      A(    ;
      A     T    109;
      A     T    105;
      AN    I   1032.7;
      AN    M   1020.0;
      AN    M   1008.0;
      AN    M   1008.2;
      AN    M   1001.0;
      O     ;
      A(    ;
      O     I      0.7;
      O     I    180.4;
      )     ;
      AN    I   1032.0;
      )     ;
      A     M   1000.6;
      A     M   1500.6;
      AN    M   1020.3;
      AN    M   1030.0;
      AN    I   1032.5;
      =     Q   1032.6;
NETWORK
TITLE =

      A     I      0.1;
      =     Q   1032.7;
NETWORK
TITLE =

      A     I      0.0;
      A     M   1000.2;
      =     Q   1033.0;
NETWORK
TITLE =

      A     M   1000.6;
      A(    ;
      O     DB51.DBX  200.7;
      O     M   4000.6;
      )     ;
      A     I   1032.0;
      AN    I   1032.7;
      AN    M   1020.3;
      =     Q   1033.1;
NETWORK
TITLE =

      A     M   1000.6;
      A     M   1500.6;
      =     Q   1033.2;
NETWORK
TITLE =

      A     M   1001.7;
      A     M   1002.1;
      =     Q   1033.3;
NETWORK
TITLE =

      A     I   1041.5;
      =     Q   1033.5;
NETWORK
TITLE =

      A     I   1057.6;
      =     Q   1033.6;
NETWORK
TITLE =

      A     I   1049.7;
      =     Q   1033.7;
NETWORK
TITLE =

      A(    ;
      A     I    278.1;
      A     M   1054.0;
      A     M   1054.3;
      A     M   1051.0;
      A     M   1051.6;
      A     M   1052.0;
      A     M   1052.4;
      A     M   1052.6;
      A     M   1053.0;
      A     T    122;
      A     M    244.1;
      O     ;
      A     M   1042.0;
      A     M   1042.2;
      A     M   1042.4;
      A     M   1042.6;
      A     M   1043.2;
      A     M   1043.4;
      A     M   1044.4;
      A(    ;
      O     M   1040.6;
      O     M   1041.7;
      )     ;
      A     T    123;
      A     M    244.0;
      )     ;
      A     M   1009.4;
      A     M   1006.5;
      AN    M   1001.0;
      AN    M   1008.2;
      =     Q   1034.0;
NETWORK
TITLE =

      A     M   1512.5;
      A     M   1512.6;
      A     I    369.0;
      A     I    369.1;
      AN    Q    368.3;
      AN    Q   1034.5;
      =     Q   1034.4;
NETWORK
TITLE =

      A     M   1512.5;
      A     M   1512.6;
      AN    I    369.0;
      A     I    369.1;
      AN    Q    368.3;
      AN    Q   1034.4;
      =     Q   1034.5;
NETWORK
TITLE =
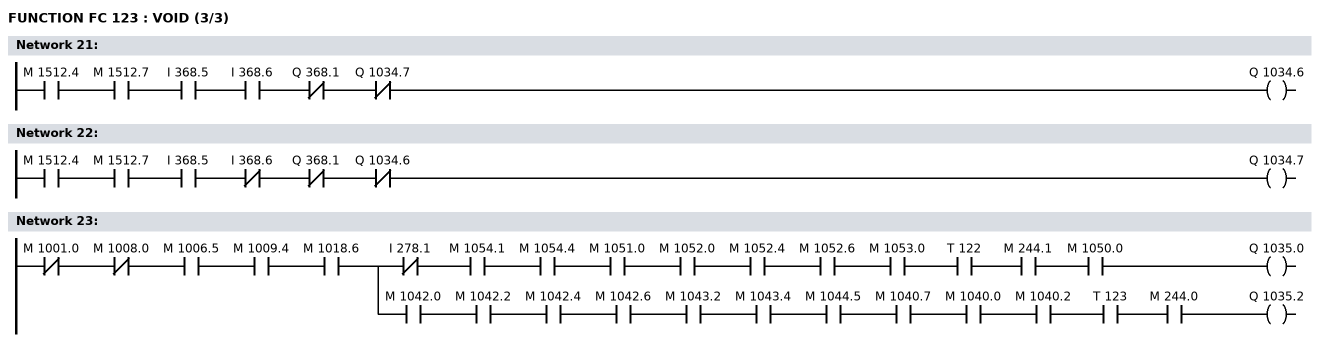

      A     M   1512.4;
      A     M   1512.7;
      A     I    368.5;
      A     I    368.6;
      AN    Q    368.1;
      AN    Q   1034.7;
      =     Q   1034.6;
NETWORK
TITLE =

      A     M   1512.4;
      A     M   1512.7;
      A     I    368.5;
      AN    I    368.6;
      AN    Q    368.1;
      AN    Q   1034.6;
      =     Q   1034.7;
NETWORK
TITLE =

      AN    M   1001.0;
      AN    M   1008.0;
      A     M   1006.5;
      A     M   1009.4;
      A     M   1018.6;
      =     L      0.0;
      A     L      0.0;
      AN    I    278.1;
      A     M   1054.1;
      A     M   1054.4;
      A     M   1051.0;
      A     M   1052.0;
      A     M   1052.4;
      A     M   1052.6;
      A     M   1053.0;
      A     T    122;
      A     M    244.1;
      A     M   1050.0;
      =     Q   1035.0;
      A     L      0.0;
      A     M   1042.0;
      A     M   1042.2;
      A     M   1042.4;
      A     M   1042.6;
      A     M   1043.2;
      A     M   1043.4;
      A     M   1044.5;
      A     M   1040.7;
      A     M   1040.0;
      A     M   1040.2;
      A     T    123;
      A     M    244.0;
      =     Q   1035.2;
END_FUNCTION

FUNCTION FC 124 : VOID
TITLE =
VERSION : 0.1

BEGIN
NETWORK
TITLE =
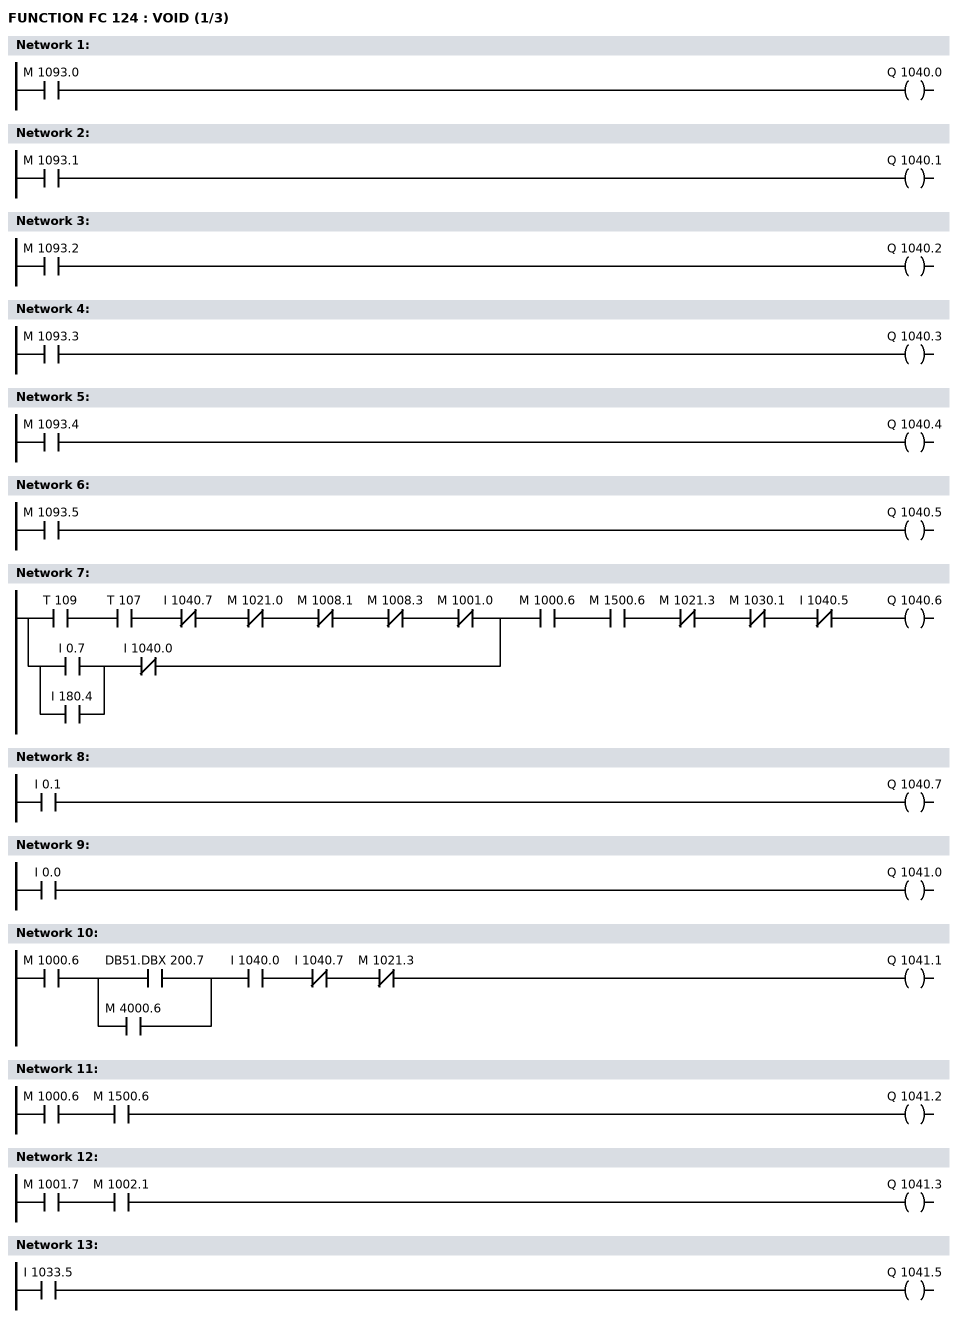

      A     M   1093.0;
      =     Q   1040.0;
NETWORK
TITLE =

      A     M   1093.1;
      =     Q   1040.1;
NETWORK
TITLE =

      A     M   1093.2;
      =     Q   1040.2;
NETWORK
TITLE =

      A     M   1093.3;
      =     Q   1040.3;
NETWORK
TITLE =

      A     M   1093.4;
      =     Q   1040.4;
NETWORK
TITLE =

      A     M   1093.5;
      =     Q   1040.5;
NETWORK
TITLE =

      A(    ;
      A     T    109;
      A     T    107;
      AN    I   1040.7;
      AN    M   1021.0;
      AN    M   1008.1;
      AN    M   1008.3;
      AN    M   1001.0;
      O     ;
      A(    ;
      O     I      0.7;
      O     I    180.4;
      )     ;
      AN    I   1040.0;
      )     ;
      A     M   1000.6;
      A     M   1500.6;
      AN    M   1021.3;
      AN    M   1030.1;
      AN    I   1040.5;
      =     Q   1040.6;
NETWORK
TITLE =

      A     I      0.1;
      =     Q   1040.7;
NETWORK
TITLE =

      A     I      0.0;
      =     Q   1041.0;
NETWORK
TITLE =

      A     M   1000.6;
      A(    ;
      O     DB51.DBX  200.7;
      O     M   4000.6;
      )     ;
      A     I   1040.0;
      AN    I   1040.7;
      AN    M   1021.3;
      =     Q   1041.1;
NETWORK
TITLE =

      A     M   1000.6;
      A     M   1500.6;
      =     Q   1041.2;
NETWORK
TITLE =

      A     M   1001.7;
      A     M   1002.1;
      =     Q   1041.3;
NETWORK
TITLE =

      A     I   1033.5;
      =     Q   1041.5;
NETWORK
TITLE =
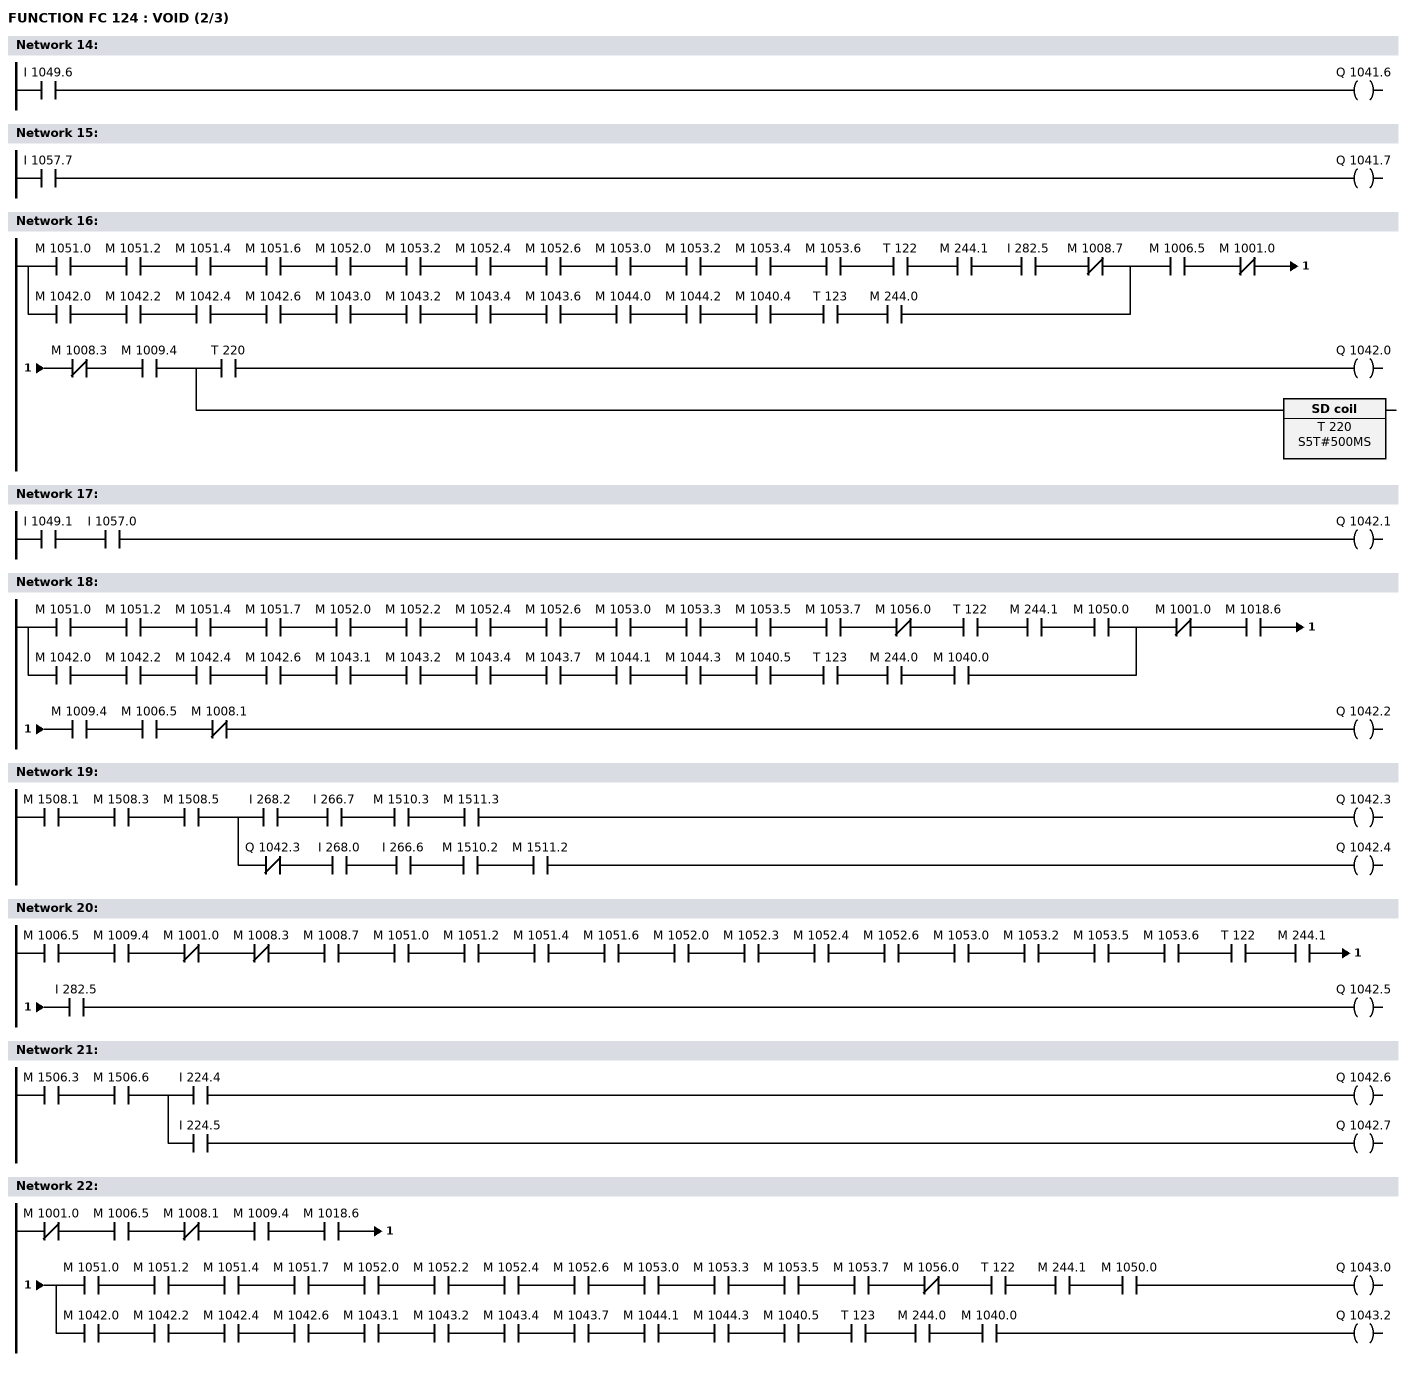

      A     I   1049.6;
      =     Q   1041.6;
NETWORK
TITLE =

      A     I   1057.7;
      =     Q   1041.7;
NETWORK
TITLE =

      A(    ;
      A     M   1051.0;
      A     M   1051.2;
      A     M   1051.4;
      A     M   1051.6;
      A     M   1052.0;
      A     M   1053.2;
      A     M   1052.4;
      A     M   1052.6;
      A     M   1053.0;
      A     M   1053.2;
      A     M   1053.4;
      A     M   1053.6;
      A     T    122;
      A     M    244.1;
      A     I    282.5;
      AN    M   1008.7;
      O     ;
      A     M   1042.0;
      A     M   1042.2;
      A     M   1042.4;
      A     M   1042.6;
      A     M   1043.0;
      A     M   1043.2;
      A     M   1043.4;
      A     M   1043.6;
      A     M   1044.0;
      A     M   1044.2;
      A     M   1040.4;
      A     T    123;
      A     M    244.0;
      )     ;
      A     M   1006.5;
      AN    M   1001.0;
      AN    M   1008.3;
      A     M   1009.4;
      =     L      0.0;
      A     L      0.0;
      A     T    220;
      =     Q   1042.0;
      A     L      0.0;
      BLD   102;
      L     S5T#500MS;
      SD    T    220;
NETWORK
TITLE =

      A     I   1049.1;
      A     I   1057.0;
      =     Q   1042.1;
NETWORK
TITLE =

      A(    ;
      A     M   1051.0;
      A     M   1051.2;
      A     M   1051.4;
      A     M   1051.7;
      A     M   1052.0;
      A     M   1052.2;
      A     M   1052.4;
      A     M   1052.6;
      A     M   1053.0;
      A     M   1053.3;
      A     M   1053.5;
      A     M   1053.7;
      AN    M   1056.0;
      A     T    122;
      A     M    244.1;
      A     M   1050.0;
      O     ;
      A     M   1042.0;
      A     M   1042.2;
      A     M   1042.4;
      A     M   1042.6;
      A     M   1043.1;
      A     M   1043.2;
      A     M   1043.4;
      A     M   1043.7;
      A     M   1044.1;
      A     M   1044.3;
      A     M   1040.5;
      A     T    123;
      A     M    244.0;
      A     M   1040.0;
      )     ;
      AN    M   1001.0;
      A     M   1018.6;
      A     M   1009.4;
      A     M   1006.5;
      AN    M   1008.1;
      =     Q   1042.2;
NETWORK
TITLE =

      A     M   1508.1;
      A     M   1508.3;
      A     M   1508.5;
      =     L      0.0;
      A     L      0.0;
      A     I    268.2;
      A     I    266.7;
      A     M   1510.3;
      A     M   1511.3;
      =     Q   1042.3;
      A     L      0.0;
      AN    Q   1042.3;
      A     I    268.0;
      A     I    266.6;
      A     M   1510.2;
      A     M   1511.2;
      =     Q   1042.4;
NETWORK
TITLE =

      A     M   1006.5;
      A     M   1009.4;
      AN    M   1001.0;
      AN    M   1008.3;
      A     M   1008.7;
      A     M   1051.0;
      A     M   1051.2;
      A     M   1051.4;
      A     M   1051.6;
      A     M   1052.0;
      A     M   1052.3;
      A     M   1052.4;
      A     M   1052.6;
      A     M   1053.0;
      A     M   1053.2;
      A     M   1053.5;
      A     M   1053.6;
      A     T    122;
      A     M    244.1;
      A     I    282.5;
      =     Q   1042.5;
NETWORK
TITLE =

      A     M   1506.3;
      A     M   1506.6;
      =     L      0.0;
      A     L      0.0;
      A     I    224.4;
      =     Q   1042.6;
      A     L      0.0;
      A     I    224.5;
      =     Q   1042.7;
NETWORK
TITLE =

      AN    M   1001.0;
      A     M   1006.5;
      AN    M   1008.1;
      A     M   1009.4;
      A     M   1018.6;
      =     L      0.0;
      A     L      0.0;
      A     M   1051.0;
      A     M   1051.2;
      A     M   1051.4;
      A     M   1051.7;
      A     M   1052.0;
      A     M   1052.2;
      A     M   1052.4;
      A     M   1052.6;
      A     M   1053.0;
      A     M   1053.3;
      A     M   1053.5;
      A     M   1053.7;
      AN    M   1056.0;
      A     T    122;
      A     M    244.1;
      A     M   1050.0;
      =     Q   1043.0;
      A     L      0.0;
      A     M   1042.0;
      A     M   1042.2;
      A     M   1042.4;
      A     M   1042.6;
      A     M   1043.1;
      A     M   1043.2;
      A     M   1043.4;
      A     M   1043.7;
      A     M   1044.1;
      A     M   1044.3;
      A     M   1040.5;
      A     T    123;
      A     M    244.0;
      A     M   1040.0;
      =     Q   1043.2;
NETWORK
TITLE =
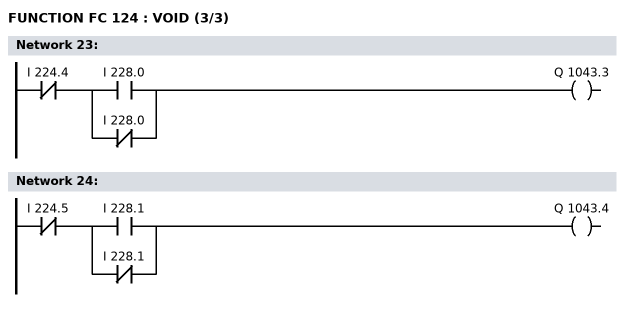

      AN    I    224.4;
      A(    ;
      O     I    228.0;
      ON    I    228.0;
      )     ;
      =     Q   1043.3;
NETWORK
TITLE =

      AN    I    224.5;
      A(    ;
      O     I    228.1;
      ON    I    228.1;
      )     ;
      =     Q   1043.4;
END_FUNCTION

FUNCTION FC 125 : VOID
TITLE =
VERSION : 0.1

BEGIN
NETWORK
TITLE =

      A     I   1048.0;
      JNB   _001;
      L     0;
      T     MB  1094;
_001: NOP   0;
NETWORK
TITLE =

      AN    OV;
      =     L      0.0;
      A     L      0.0;
      A     M    164.1;
      =     L      0.1;
      A     L      0.1;
      AN    M    167.7;
      A     I   1048.0;
      JNB   _002;
      L     11;
      T     MB  1094;
_002: NOP   0;
      A     L      0.1;
      A     M    167.7;
      A     I   1048.0;
      JNB   _003;
      L     19;
      T     MB  1094;
_003: NOP   0;
      A     L      0.0;
      A     M    164.0;
      A     I   1048.0;
      JNB   _004;
      L     1;
      T     MB  1094;
_004: NOP   0;
NETWORK
TITLE =
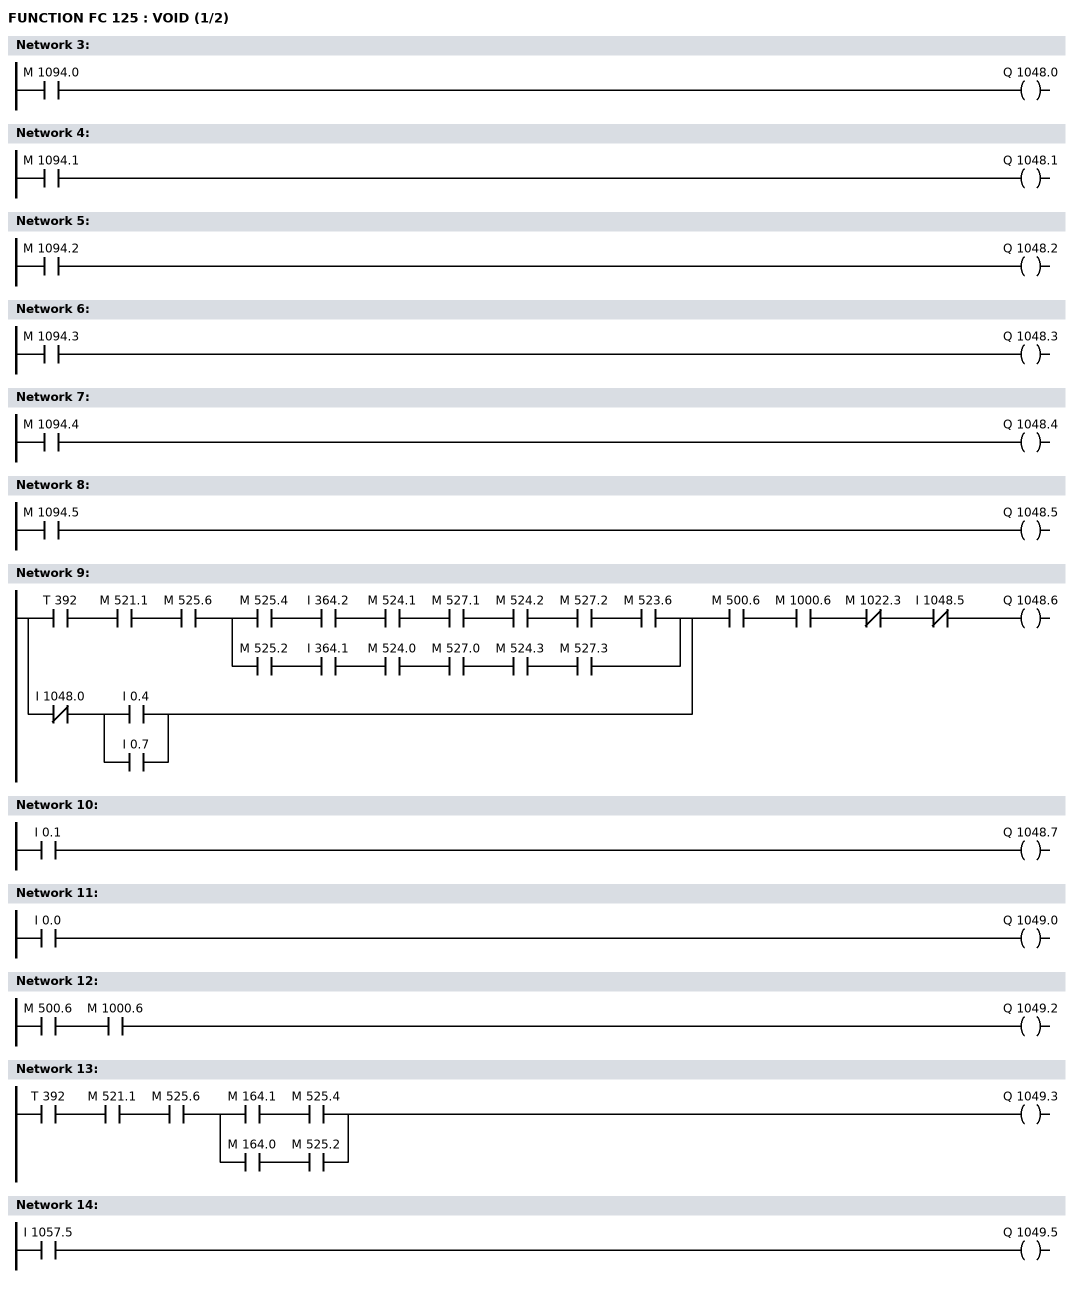

      A     M   1094.0;
      =     Q   1048.0;
NETWORK
TITLE =

      A     M   1094.1;
      =     Q   1048.1;
NETWORK
TITLE =

      A     M   1094.2;
      =     Q   1048.2;
NETWORK
TITLE =

      A     M   1094.3;
      =     Q   1048.3;
NETWORK
TITLE =

      A     M   1094.4;
      =     Q   1048.4;
NETWORK
TITLE =

      A     M   1094.5;
      =     Q   1048.5;
NETWORK
TITLE =

      A(    ;
      A     T    392;
      A     M    521.1;
      A     M    525.6;
      A(    ;
      A     M    525.4;
      A     I    364.2;
      A     M    524.1;
      A     M    527.1;
      A     M    524.2;
      A     M    527.2;
      A     M    523.6;
      O     ;
      A     M    525.2;
      A     I    364.1;
      A     M    524.0;
      A     M    527.0;
      A     M    524.3;
      A     M    527.3;
      )     ;
      O     ;
      AN    I   1048.0;
      A(    ;
      O     I      0.4;
      O     I      0.7;
      )     ;
      )     ;
      A     M    500.6;
      A     M   1000.6;
      AN    M   1022.3;
      AN    I   1048.5;
      =     Q   1048.6;
NETWORK
TITLE =

      A     I      0.1;
      =     Q   1048.7;
NETWORK
TITLE =

      A     I      0.0;
      =     Q   1049.0;
NETWORK
TITLE =

      A     M    500.6;
      A     M   1000.6;
      =     Q   1049.2;
NETWORK
TITLE =

      A     T    392;
      A     M    521.1;
      A     M    525.6;
      A(    ;
      A     M    164.1;
      A     M    525.4;
      O     ;
      A     M    164.0;
      A     M    525.2;
      )     ;
      =     Q   1049.3;
NETWORK
TITLE =

      A     I   1057.5;
      =     Q   1049.5;
NETWORK
TITLE =
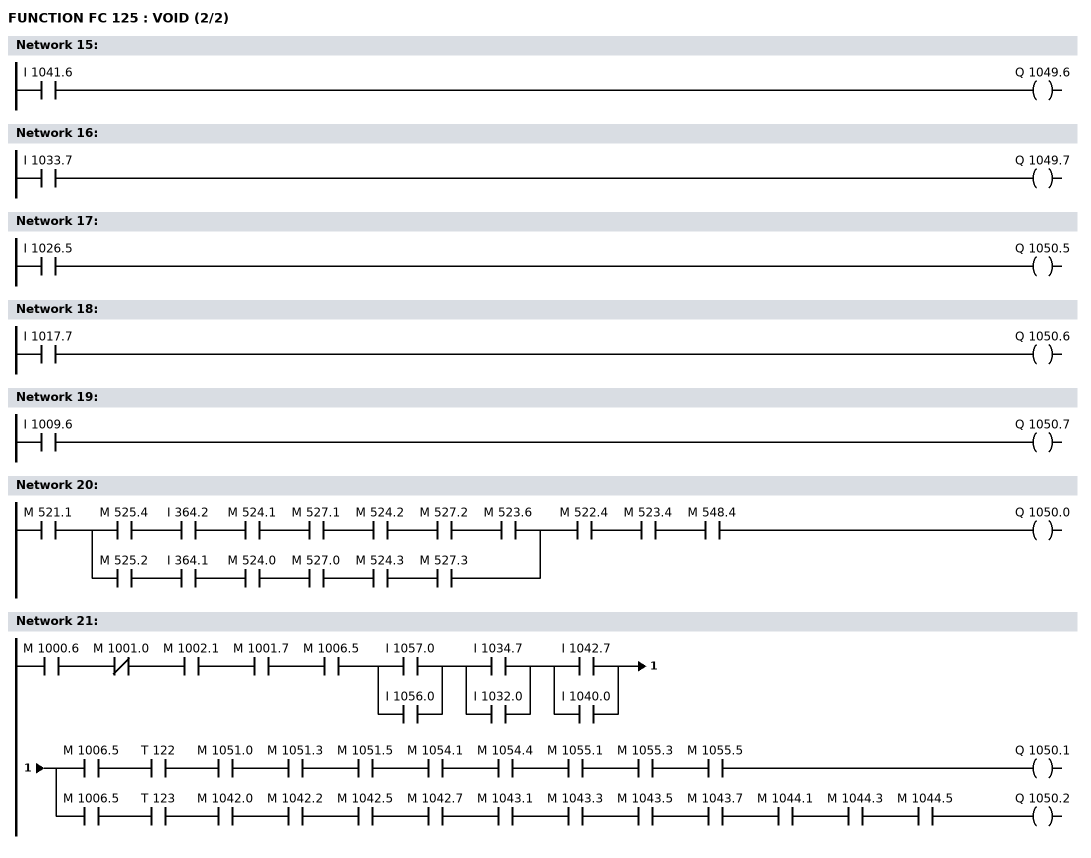

      A     I   1041.6;
      =     Q   1049.6;
NETWORK
TITLE =

      A     I   1033.7;
      =     Q   1049.7;
NETWORK
TITLE =

      A     I   1026.5;
      =     Q   1050.5;
NETWORK
TITLE =

      A     I   1017.7;
      =     Q   1050.6;
NETWORK
TITLE =

      A     I   1009.6;
      =     Q   1050.7;
NETWORK
TITLE =

      A     M    521.1;
      A(    ;
      A     M    525.4;
      A     I    364.2;
      A     M    524.1;
      A     M    527.1;
      A     M    524.2;
      A     M    527.2;
      A     M    523.6;
      O     ;
      A     M    525.2;
      A     I    364.1;
      A     M    524.0;
      A     M    527.0;
      A     M    524.3;
      A     M    527.3;
      )     ;
      A     M    522.4;
      A     M    523.4;
      A     M    548.4;
      =     Q   1050.0;
NETWORK
TITLE =

      A     M   1000.6;
      AN    M   1001.0;
      A     M   1002.1;
      A     M   1001.7;
      A     M   1006.5;
      A(    ;
      O     I   1057.0;
      O     I   1056.0;
      )     ;
      A(    ;
      O     I   1034.7;
      O     I   1032.0;
      )     ;
      A(    ;
      O     I   1042.7;
      O     I   1040.0;
      )     ;
      =     L      0.0;
      A     L      0.0;
      A     M   1006.5;
      A     T    122;
      A     M   1051.0;
      A     M   1051.3;
      A     M   1051.5;
      A     M   1054.1;
      A     M   1054.4;
      A     M   1055.1;
      A     M   1055.3;
      A     M   1055.5;
      =     Q   1050.1;
      A     L      0.0;
      A     M   1006.5;
      A     T    123;
      A     M   1042.0;
      A     M   1042.2;
      A     M   1042.5;
      A     M   1042.7;
      A     M   1043.1;
      A     M   1043.3;
      A     M   1043.5;
      A     M   1043.7;
      A     M   1044.1;
      A     M   1044.3;
      A     M   1044.5;
      =     Q   1050.2;
END_FUNCTION

FUNCTION FC 126 : VOID
TITLE =
VERSION : 0.1

BEGIN
NETWORK
TITLE =

      A(    ;
      O     I   1056.0;
      O     I   1056.1;
      )     ;
      JNB   _001;
      L     0;
      T     MB  1096;
_001: NOP   0;
NETWORK
TITLE =

      AN    OV;
      =     L      0.0;
      A     L      0.0;
      A     M    204.1;
      =     L      0.1;
      A     L      0.1;
      AN    M    207.7;
      A     I   1056.0;
      JNB   _002;
      L     11;
      T     MB  1096;
_002: NOP   0;
      A     L      0.1;
      A     M    207.7;
      A     I   1056.0;
      JNB   _003;
      L     19;
      T     MB  1096;
_003: NOP   0;
      A     L      0.0;
      A     M    204.0;
      A     I   1056.0;
      JNB   _004;
      L     1;
      T     MB  1096;
_004: NOP   0;
NETWORK
TITLE =
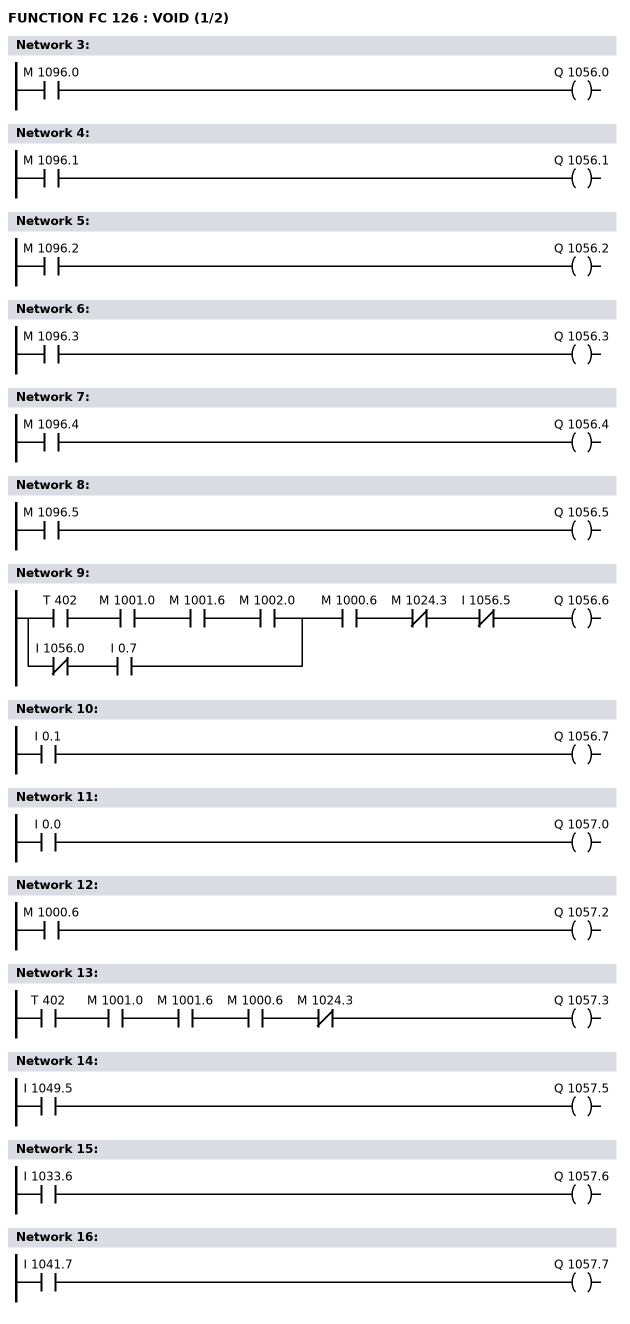

      A     M   1096.0;
      =     Q   1056.0;
NETWORK
TITLE =

      A     M   1096.1;
      =     Q   1056.1;
NETWORK
TITLE =

      A     M   1096.2;
      =     Q   1056.2;
NETWORK
TITLE =

      A     M   1096.3;
      =     Q   1056.3;
NETWORK
TITLE =

      A     M   1096.4;
      =     Q   1056.4;
NETWORK
TITLE =

      A     M   1096.5;
      =     Q   1056.5;
NETWORK
TITLE =

      A(    ;
      A     T    402;
      A     M   1001.0;
      A     M   1001.6;
      A     M   1002.0;
      O     ;
      AN    I   1056.0;
      A     I      0.7;
      )     ;
      A     M   1000.6;
      AN    M   1024.3;
      AN    I   1056.5;
      =     Q   1056.6;
NETWORK
TITLE =

      A     I      0.1;
      =     Q   1056.7;
NETWORK
TITLE =

      A     I      0.0;
      =     Q   1057.0;
NETWORK
TITLE =

      A     M   1000.6;
      =     Q   1057.2;
NETWORK
TITLE =

      A     T    402;
      A     M   1001.0;
      A     M   1001.6;
      A     M   1000.6;
      AN    M   1024.3;
      =     Q   1057.3;
NETWORK
TITLE =

      A     I   1049.5;
      =     Q   1057.5;
NETWORK
TITLE =

      A     I   1033.6;
      =     Q   1057.6;
NETWORK
TITLE =

      A     I   1041.7;
      =     Q   1057.7;
NETWORK
TITLE =
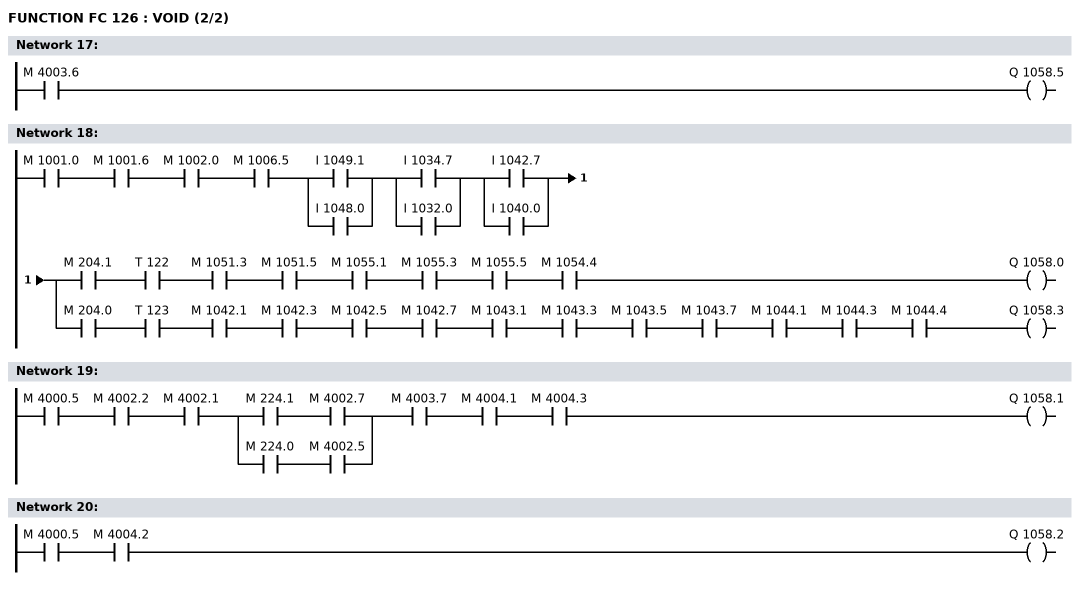

      A     M   4003.6;
      =     Q   1058.5;
NETWORK
TITLE =

      A     M   1001.0;
      A     M   1001.6;
      A     M   1002.0;
      A     M   1006.5;
      A(    ;
      O     I   1049.1;
      O     I   1048.0;
      )     ;
      A(    ;
      O     I   1034.7;
      O     I   1032.0;
      )     ;
      A(    ;
      O     I   1042.7;
      O     I   1040.0;
      )     ;
      =     L      0.0;
      A     L      0.0;
      A     M    204.1;
      A     T    122;
      A     M   1051.3;
      A     M   1051.5;
      A     M   1055.1;
      A     M   1055.3;
      A     M   1055.5;
      A     M   1054.4;
      =     Q   1058.0;
      A     L      0.0;
      A     M    204.0;
      A     T    123;
      A     M   1042.1;
      A     M   1042.3;
      A     M   1042.5;
      A     M   1042.7;
      A     M   1043.1;
      A     M   1043.3;
      A     M   1043.5;
      A     M   1043.7;
      A     M   1044.1;
      A     M   1044.3;
      A     M   1044.4;
      =     Q   1058.3;
NETWORK
TITLE =

      A     M   4000.5;
      A     M   4002.2;
      A     M   4002.1;
      A(    ;
      A     M    224.1;
      A     M   4002.7;
      O     ;
      A     M    224.0;
      A     M   4002.5;
      )     ;
      A     M   4003.7;
      A     M   4004.1;
      A     M   4004.3;
      =     Q   1058.1;
NETWORK
TITLE =

      A     M   4000.5;
      A     M   4004.2;
      =     Q   1058.2;
END_FUNCTION

FUNCTION_BLOCK FB 130
TITLE =
VERSION : 0.1


VAR
  EXTN_STN_MODE : FB 402;	//EXTN_STN_MODE
END_VAR
BEGIN
NETWORK
TITLE =
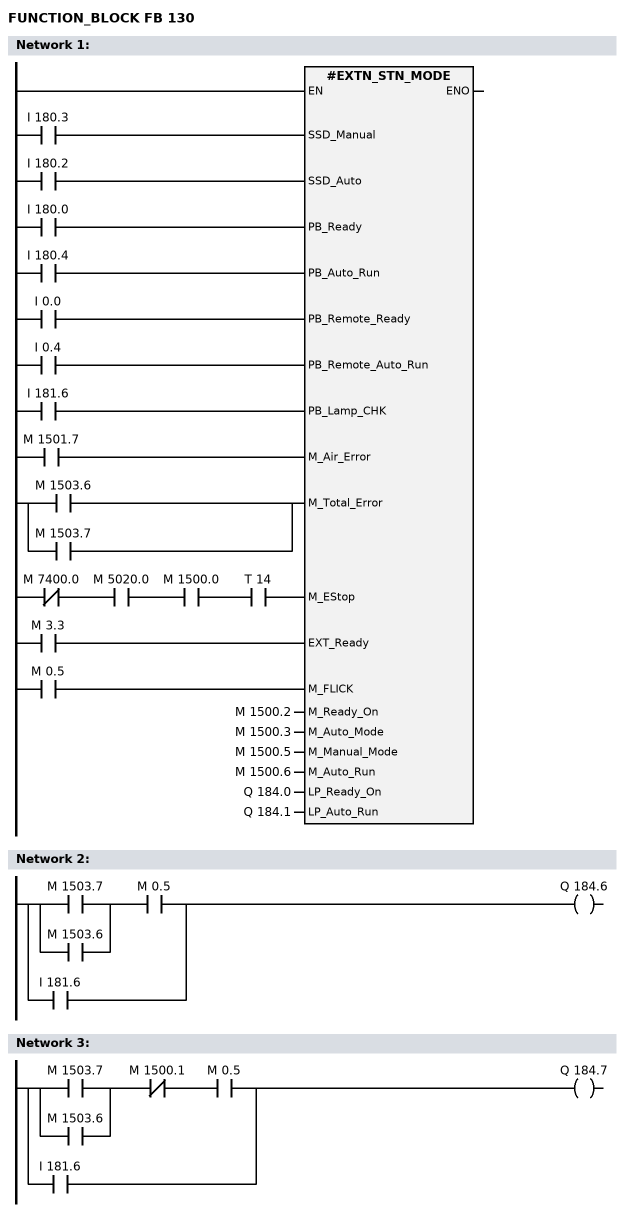

      A     I    180.3;
      =     L      0.0;
      BLD   103;
      A     I    180.2;
      =     L      0.1;
      BLD   103;
      A     I    180.0;
      =     L      0.2;
      BLD   103;
      A     I    180.4;
      =     L      0.3;
      BLD   103;
      A     I      0.0;
      =     L      0.4;
      BLD   103;
      A     I      0.4;
      =     L      0.5;
      BLD   103;
      A     I    181.6;
      =     L      0.6;
      BLD   103;
      A     M   1501.7;
      =     L      0.7;
      BLD   103;
      A(    ;
      O     M   1503.6;
      O     M   1503.7;
      )     ;
      =     L      1.1;
      BLD   103;
      AN    M   7400.0;
      A     M   5020.0;
      A     M   1500.0;
      A     T     14;
      =     L      1.2;
      BLD   103;
      A     M      3.3;
      =     L      1.3;
      BLD   103;
      A     M      0.5;
      =     L      1.5;
      BLD   103;
      CALL #EXTN_STN_MODE (
           SSD_Manual               := L      0.0,
           SSD_Auto                 := L      0.1,
           PB_Ready                 := L      0.2,
           PB_Auto_Run              := L      0.3,
           PB_Remote_Ready          := L      0.4,
           PB_Remote_Auto_Run       := L      0.5,
           PB_Lamp_CHK              := L      0.6,
           M_Air_Error              := L      0.7,
           M_Total_Error            := L      1.1,
           M_EStop                  := L      1.2,
           EXT_Ready                := L      1.3,
           M_FLICK                  := L      1.5,
           M_Ready_On               := M   1500.2,
           M_Auto_Mode              := M   1500.3,
           M_Manual_Mode            := M   1500.5,
           M_Auto_Run               := M   1500.6,
           LP_Ready_On              := Q    184.0,
           LP_Auto_Run              := Q    184.1);
      NOP   0;
NETWORK
TITLE =

      A(    ;
      O     M   1503.7;
      O     M   1503.6;
      )     ;
      A     M      0.5;
      O     I    181.6;
      =     Q    184.6;
NETWORK
TITLE =

      A(    ;
      O     M   1503.7;
      O     M   1503.6;
      )     ;
      AN    M   1500.1;
      A     M      0.5;
      O     I    181.6;
      =     Q    184.7;
END_FUNCTION_BLOCK

DATA_BLOCK DB 130
TITLE =
VERSION : 0.0

 FB 130
BEGIN
   EXTN_STN_MODE.SSD_Manual := FALSE;
   EXTN_STN_MODE.SSD_Auto := FALSE;
   EXTN_STN_MODE.PB_Ready := FALSE;
   EXTN_STN_MODE.PB_Auto_Run := FALSE;
   EXTN_STN_MODE.PB_Remote_Ready := FALSE;
   EXTN_STN_MODE.PB_Remote_Auto_Run := FALSE;
   EXTN_STN_MODE.PB_Lamp_CHK := FALSE;
   EXTN_STN_MODE.M_Air_Error := FALSE;
   EXTN_STN_MODE.M_Water_Error := FALSE;
   EXTN_STN_MODE.M_Total_Error := FALSE;
   EXTN_STN_MODE.M_EStop := FALSE;
   EXTN_STN_MODE.EXT_Ready := FALSE;
   EXTN_STN_MODE.EXT_Auto := FALSE;
   EXTN_STN_MODE.T_SemiAuto := T#0MS;
   EXTN_STN_MODE.M_FLICK := FALSE;
   EXTN_STN_MODE.M_Ready_On := FALSE;
   EXTN_STN_MODE.M_Auto_Mode := FALSE;
   EXTN_STN_MODE.M_SemiAuto_Mode := FALSE;
   EXTN_STN_MODE.M_Manual_Mode := FALSE;
   EXTN_STN_MODE.M_Auto_Run := FALSE;
   EXTN_STN_MODE.LP_Ready_On := FALSE;
   EXTN_STN_MODE.LP_Auto_Run := FALSE;
   EXTN_STN_MODE.AUTO_MODE_DELAY.IN := FALSE;
   EXTN_STN_MODE.AUTO_MODE_DELAY.PT := T#0MS;
   EXTN_STN_MODE.AUTO_MODE_DELAY.Q := FALSE;
   EXTN_STN_MODE.AUTO_MODE_DELAY.ET := T#0MS;
   EXTN_STN_MODE.AUTO_MODE_DELAY.STATE := B#16#0;
   EXTN_STN_MODE.AUTO_MODE_DELAY.STIME := T#0MS;
   EXTN_STN_MODE.AUTO_MODE_DELAY.ATIME := T#0MS;
   EXTN_STN_MODE.SEMI_AUTO_DELAY.IN := FALSE;
   EXTN_STN_MODE.SEMI_AUTO_DELAY.PT := T#0MS;
   EXTN_STN_MODE.SEMI_AUTO_DELAY.Q := FALSE;
   EXTN_STN_MODE.SEMI_AUTO_DELAY.ET := T#0MS;
   EXTN_STN_MODE.SEMI_AUTO_DELAY.STATE := B#16#0;
   EXTN_STN_MODE.SEMI_AUTO_DELAY.STIME := T#0MS;
   EXTN_STN_MODE.SEMI_AUTO_DELAY.ATIME := T#0MS;
   EXTN_STN_MODE.MANUAL_DELAY.IN := FALSE;
   EXTN_STN_MODE.MANUAL_DELAY.PT := T#0MS;
   EXTN_STN_MODE.MANUAL_DELAY.Q := FALSE;
   EXTN_STN_MODE.MANUAL_DELAY.ET := T#0MS;
   EXTN_STN_MODE.MANUAL_DELAY.STATE := B#16#0;
   EXTN_STN_MODE.MANUAL_DELAY.STIME := T#0MS;
   EXTN_STN_MODE.MANUAL_DELAY.ATIME := T#0MS;
END_DATA_BLOCK

FUNCTION FC 130 : VOID
TITLE =
VERSION : 0.1

BEGIN
NETWORK
TITLE =
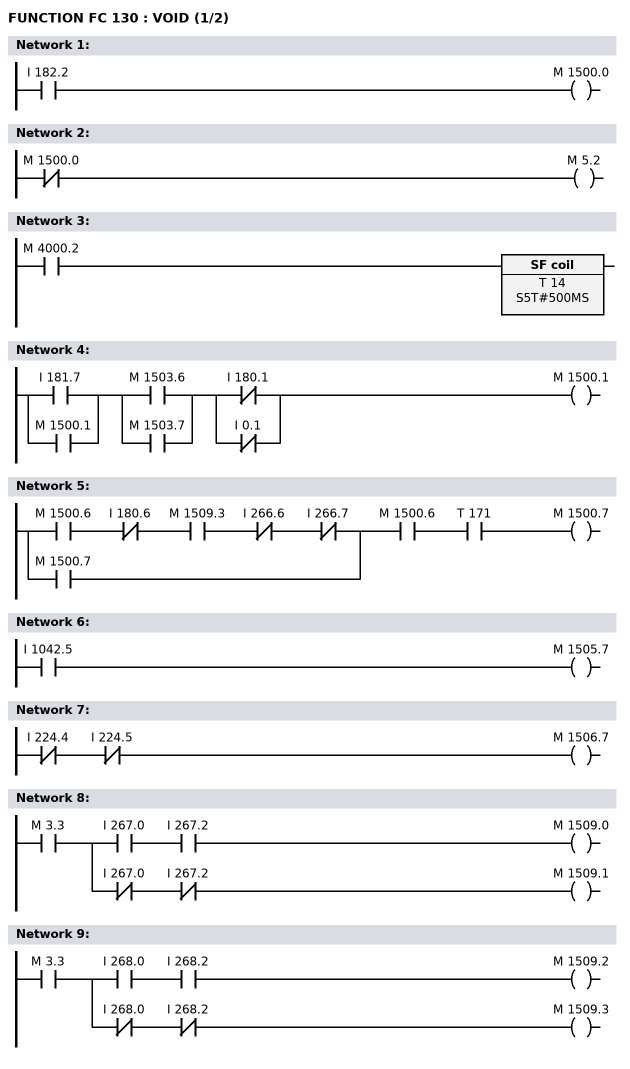

      A     I    182.2;
      =     M   1500.0;
NETWORK
TITLE =

      AN    M   1500.0;
      =     M      5.2;
NETWORK
TITLE =

      A     M   4000.2;
      L     S5T#500MS;
      SF    T     14;
NETWORK
TITLE =

      A(    ;
      O     I    181.7;
      O     M   1500.1;
      )     ;
      A(    ;
      O     M   1503.6;
      O     M   1503.7;
      )     ;
      A(    ;
      ON    I    180.1;
      ON    I      0.1;
      )     ;
      =     M   1500.1;
NETWORK
TITLE =

      A(    ;
      A     M   1500.6;
      AN    I    180.6;
      A     M   1509.3;
      AN    I    266.6;
      AN    I    266.7;
      O     M   1500.7;
      )     ;
      A     M   1500.6;
      A     T    171;
      =     M   1500.7;
NETWORK
TITLE =

      A     I   1042.5;
      =     M   1505.7;
NETWORK
TITLE =

      AN    I    224.4;
      AN    I    224.5;
      =     M   1506.7;
NETWORK
TITLE =

      A     M      3.3;
      =     L      0.0;
      A     L      0.0;
      A     I    267.0;
      A     I    267.2;
      =     M   1509.0;
      A     L      0.0;
      AN    I    267.0;
      AN    I    267.2;
      =     M   1509.1;
NETWORK
TITLE =

      A     M      3.3;
      =     L      0.0;
      A     L      0.0;
      A     I    268.0;
      A     I    268.2;
      =     M   1509.2;
      A     L      0.0;
      AN    I    268.0;
      AN    I    268.2;
      =     M   1509.3;
NETWORK
TITLE =
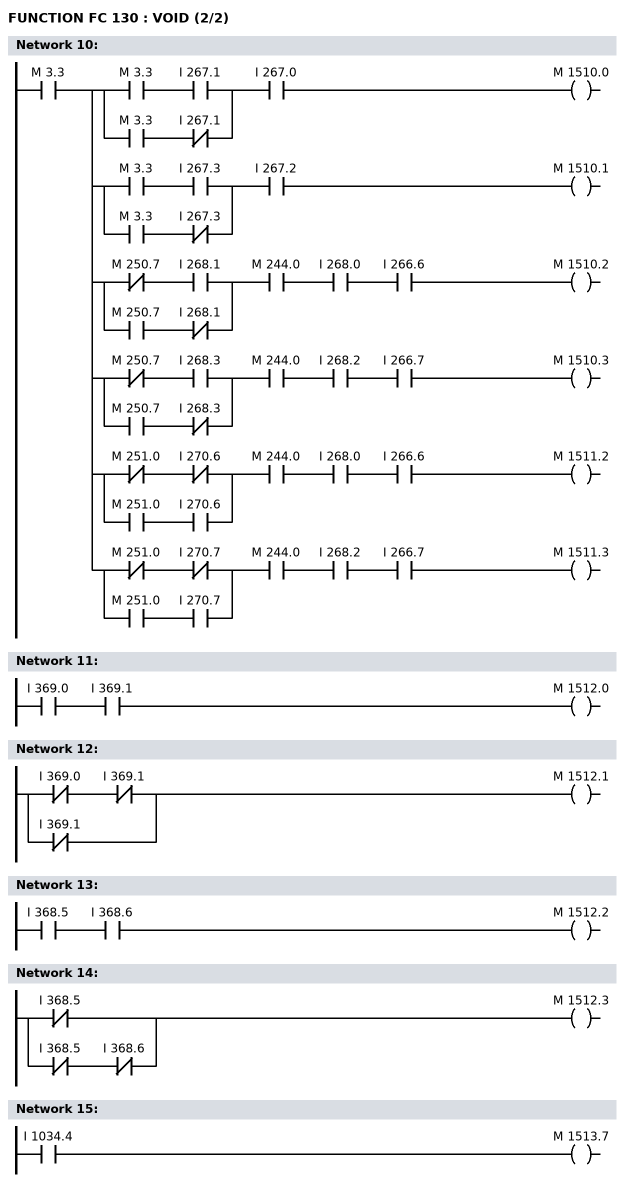

      A     M      3.3;
      =     L      0.0;
      A     L      0.0;
      A(    ;
      A     M      3.3;
      A     I    267.1;
      O     ;
      A     M      3.3;
      AN    I    267.1;
      )     ;
      A     I    267.0;
      =     M   1510.0;
      A     L      0.0;
      A(    ;
      A     M      3.3;
      A     I    267.3;
      O     ;
      A     M      3.3;
      AN    I    267.3;
      )     ;
      A     I    267.2;
      =     M   1510.1;
      A     L      0.0;
      A(    ;
      AN    M    250.7;
      A     I    268.1;
      O     ;
      A     M    250.7;
      AN    I    268.1;
      )     ;
      A     M    244.0;
      A     I    268.0;
      A     I    266.6;
      =     M   1510.2;
      A     L      0.0;
      A(    ;
      AN    M    250.7;
      A     I    268.3;
      O     ;
      A     M    250.7;
      AN    I    268.3;
      )     ;
      A     M    244.0;
      A     I    268.2;
      A     I    266.7;
      =     M   1510.3;
      A     L      0.0;
      A(    ;
      AN    M    251.0;
      AN    I    270.6;
      O     ;
      A     M    251.0;
      A     I    270.6;
      )     ;
      A     M    244.0;
      A     I    268.0;
      A     I    266.6;
      =     M   1511.2;
      A     L      0.0;
      A(    ;
      AN    M    251.0;
      AN    I    270.7;
      O     ;
      A     M    251.0;
      A     I    270.7;
      )     ;
      A     M    244.0;
      A     I    268.2;
      A     I    266.7;
      =     M   1511.3;
NETWORK
TITLE =

      A     I    369.0;
      A     I    369.1;
      =     M   1512.0;
NETWORK
TITLE =

      AN    I    369.0;
      AN    I    369.1;
      ON    I    369.1;
      =     M   1512.1;
NETWORK
TITLE =

      A     I    368.5;
      A     I    368.6;
      =     M   1512.2;
NETWORK
TITLE =

      ON    I    368.5;
      O     ;
      AN    I    368.5;
      AN    I    368.6;
      =     M   1512.3;
NETWORK
TITLE =

      A     I   1034.4;
      =     M   1513.7;
END_FUNCTION

FUNCTION_BLOCK FB 131
TITLE =
VERSION : 0.1


VAR
  S701_FDR_A_STORAGE_ERR : FB 424;
  S701_FDR_B_STORAGE_ERR : FB 424;
  LM_EXTN_UNIT_ERR : FB 426;
  LM_EXTN_ADV_RET_ERR : FB 424;
  TL_EXTN_UNIT_ERR : FB 426;
  TL_EXTN_ADV_RET_ERR : FB 424;
END_VAR
BEGIN
NETWORK
TITLE =
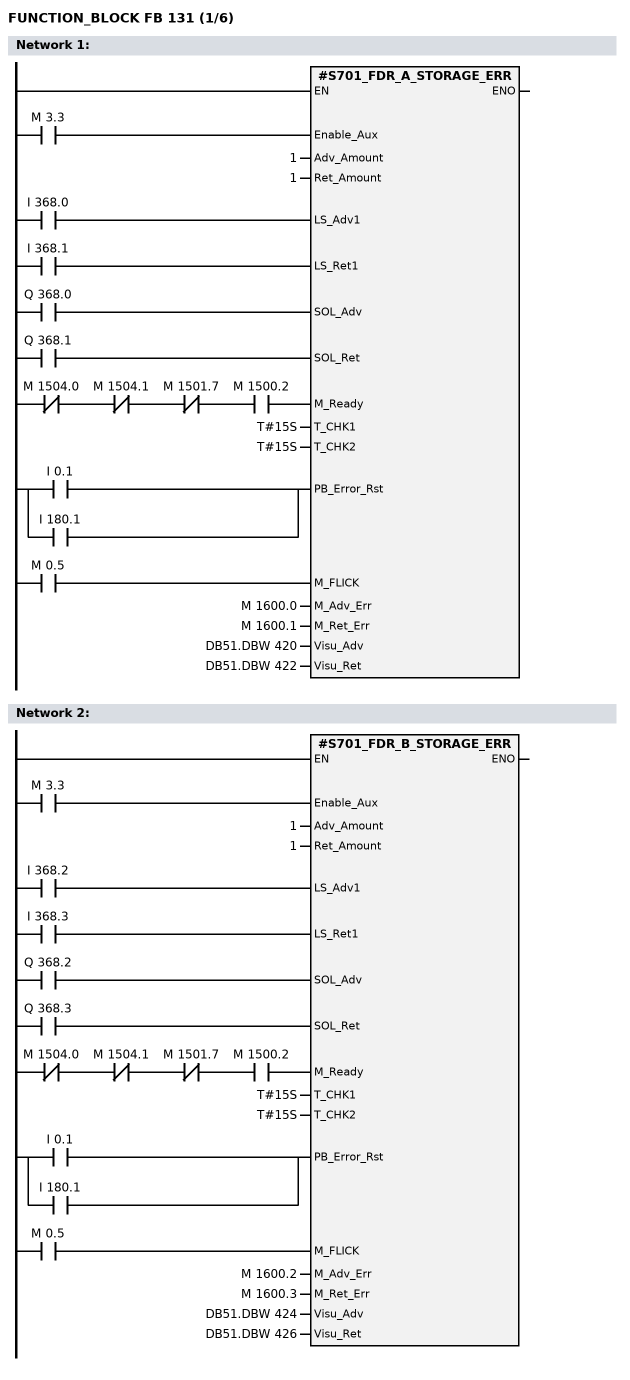

      A     M      3.3;
      =     L      0.0;
      BLD   103;
      A     I    368.0;
      =     L      0.1;
      BLD   103;
      A     I    368.1;
      =     L      0.2;
      BLD   103;
      A     Q    368.0;
      =     L      1.1;
      BLD   103;
      A     Q    368.1;
      =     L      1.2;
      BLD   103;
      AN    M   1504.0;
      AN    M   1504.1;
      AN    M   1501.7;
      A     M   1500.2;
      =     L      1.3;
      BLD   103;
      A(    ;
      O     I      0.1;
      O     I    180.1;
      )     ;
      =     L      1.5;
      BLD   103;
      A     M      0.5;
      =     L      1.6;
      BLD   103;
      CALL #S701_FDR_A_STORAGE_ERR (
           Enable_Aux               := L      0.0,
           Adv_Amount               := 1,
           Ret_Amount               := 1,
           LS_Adv1                  := L      0.1,
           LS_Ret1                  := L      0.2,
           SOL_Adv                  := L      1.1,
           SOL_Ret                  := L      1.2,
           M_Ready                  := L      1.3,
           T_CHK1                   := T#15S,
           T_CHK2                   := T#15S,
           PB_Error_Rst             := L      1.5,
           M_FLICK                  := L      1.6,
           M_Adv_Err                := M   1600.0,
           M_Ret_Err                := M   1600.1,
           Visu_Adv                 := DB51.DBW  420,
           Visu_Ret                 := DB51.DBW  422);
      NOP   0;
NETWORK
TITLE =

      A     M      3.3;
      =     L      0.0;
      BLD   103;
      A     I    368.2;
      =     L      0.1;
      BLD   103;
      A     I    368.3;
      =     L      0.2;
      BLD   103;
      A     Q    368.2;
      =     L      1.1;
      BLD   103;
      A     Q    368.3;
      =     L      1.2;
      BLD   103;
      AN    M   1504.0;
      AN    M   1504.1;
      AN    M   1501.7;
      A     M   1500.2;
      =     L      1.3;
      BLD   103;
      A(    ;
      O     I      0.1;
      O     I    180.1;
      )     ;
      =     L      1.5;
      BLD   103;
      A     M      0.5;
      =     L      1.6;
      BLD   103;
      CALL #S701_FDR_B_STORAGE_ERR (
           Enable_Aux               := L      0.0,
           Adv_Amount               := 1,
           Ret_Amount               := 1,
           LS_Adv1                  := L      0.1,
           LS_Ret1                  := L      0.2,
           SOL_Adv                  := L      1.1,
           SOL_Ret                  := L      1.2,
           M_Ready                  := L      1.3,
           T_CHK1                   := T#15S,
           T_CHK2                   := T#15S,
           PB_Error_Rst             := L      1.5,
           M_FLICK                  := L      1.6,
           M_Adv_Err                := M   1600.2,
           M_Ret_Err                := M   1600.3,
           Visu_Adv                 := DB51.DBW  424,
           Visu_Ret                 := DB51.DBW  426);
      NOP   0;
NETWORK
TITLE =
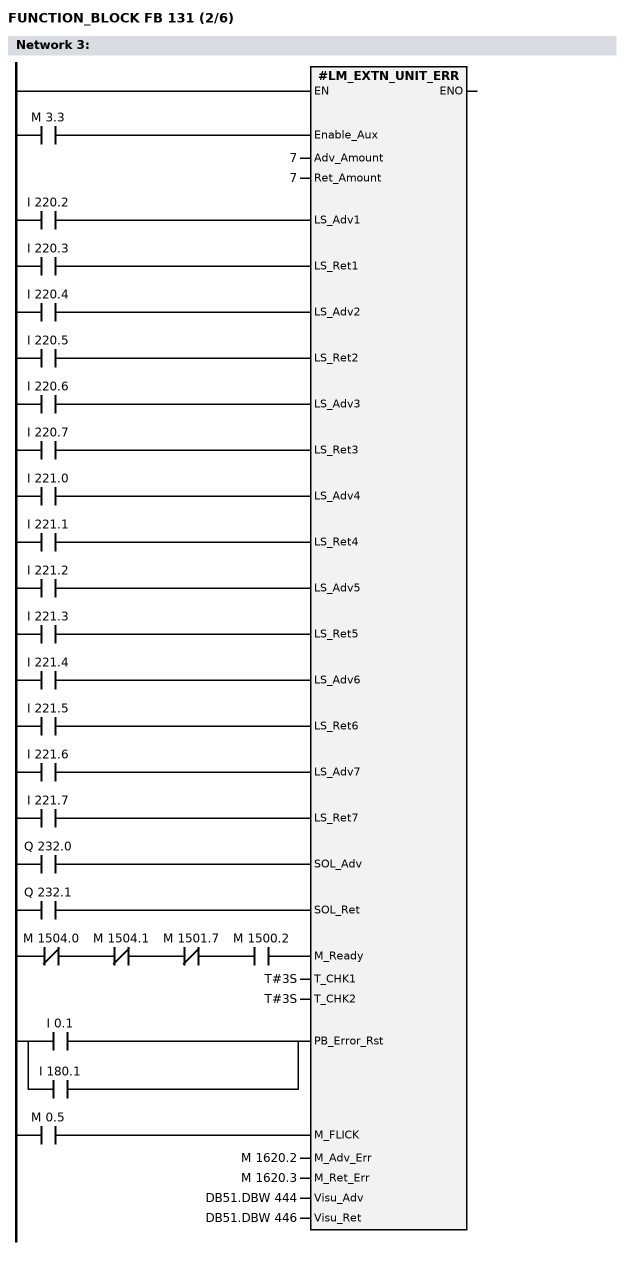

      A     M      3.3;
      =     L      0.0;
      BLD   103;
      A     I    220.2;
      =     L      0.1;
      BLD   103;
      A     I    220.3;
      =     L      0.2;
      BLD   103;
      A     I    220.4;
      =     L      0.3;
      BLD   103;
      A     I    220.5;
      =     L      0.4;
      BLD   103;
      A     I    220.6;
      =     L      0.5;
      BLD   103;
      A     I    220.7;
      =     L      0.6;
      BLD   103;
      A     I    221.0;
      =     L      0.7;
      BLD   103;
      A     I    221.1;
      =     L      1.0;
      BLD   103;
      A     I    221.2;
      =     L      1.1;
      BLD   103;
      A     I    221.3;
      =     L      1.2;
      BLD   103;
      A     I    221.4;
      =     L      1.3;
      BLD   103;
      A     I    221.5;
      =     L      1.4;
      BLD   103;
      A     I    221.6;
      =     L      1.5;
      BLD   103;
      A     I    221.7;
      =     L      1.6;
      BLD   103;
      A     Q    232.0;
      =     L      2.1;
      BLD   103;
      A     Q    232.1;
      =     L      2.2;
      BLD   103;
      AN    M   1504.0;
      AN    M   1504.1;
      AN    M   1501.7;
      A     M   1500.2;
      =     L      2.3;
      BLD   103;
      A(    ;
      O     I      0.1;
      O     I    180.1;
      )     ;
      =     L      2.5;
      BLD   103;
      A     M      0.5;
      =     L      2.6;
      BLD   103;
      CALL #LM_EXTN_UNIT_ERR (
           Enable_Aux               := L      0.0,
           Adv_Amount               := 7,
           Ret_Amount               := 7,
           LS_Adv1                  := L      0.1,
           LS_Ret1                  := L      0.2,
           LS_Adv2                  := L      0.3,
           LS_Ret2                  := L      0.4,
           LS_Adv3                  := L      0.5,
           LS_Ret3                  := L      0.6,
           LS_Adv4                  := L      0.7,
           LS_Ret4                  := L      1.0,
           LS_Adv5                  := L      1.1,
           LS_Ret5                  := L      1.2,
           LS_Adv6                  := L      1.3,
           LS_Ret6                  := L      1.4,
           LS_Adv7                  := L      1.5,
           LS_Ret7                  := L      1.6,
           SOL_Adv                  := L      2.1,
           SOL_Ret                  := L      2.2,
           M_Ready                  := L      2.3,
           T_CHK1                   := T#3S,
           T_CHK2                   := T#3S,
           PB_Error_Rst             := L      2.5,
           M_FLICK                  := L      2.6,
           M_Adv_Err                := M   1620.2,
           M_Ret_Err                := M   1620.3,
           Visu_Adv                 := DB51.DBW  444,
           Visu_Ret                 := DB51.DBW  446);
      NOP   0;
NETWORK
TITLE =
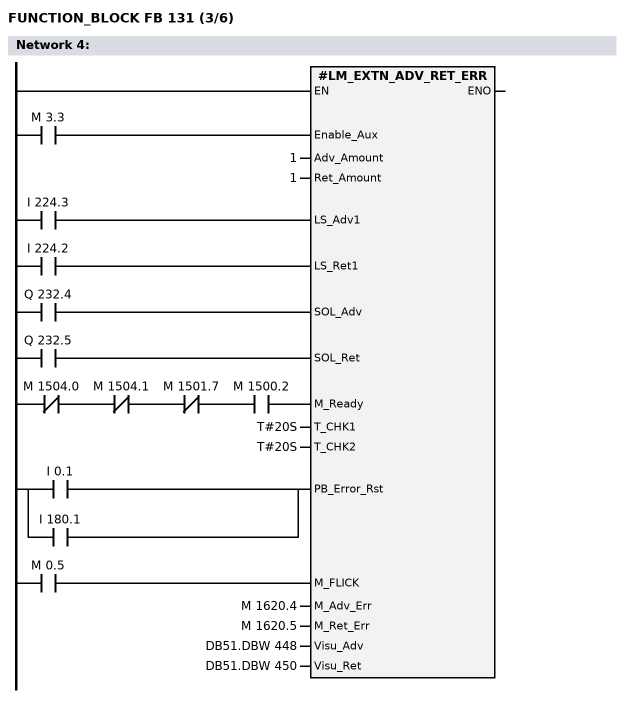

      A     M      3.3;
      =     L      0.0;
      BLD   103;
      A     I    224.3;
      =     L      0.1;
      BLD   103;
      A     I    224.2;
      =     L      0.2;
      BLD   103;
      A     Q    232.4;
      =     L      1.1;
      BLD   103;
      A     Q    232.5;
      =     L      1.2;
      BLD   103;
      AN    M   1504.0;
      AN    M   1504.1;
      AN    M   1501.7;
      A     M   1500.2;
      =     L      1.3;
      BLD   103;
      A(    ;
      O     I      0.1;
      O     I    180.1;
      )     ;
      =     L      1.5;
      BLD   103;
      A     M      0.5;
      =     L      1.6;
      BLD   103;
      CALL #LM_EXTN_ADV_RET_ERR (
           Enable_Aux               := L      0.0,
           Adv_Amount               := 1,
           Ret_Amount               := 1,
           LS_Adv1                  := L      0.1,
           LS_Ret1                  := L      0.2,
           SOL_Adv                  := L      1.1,
           SOL_Ret                  := L      1.2,
           M_Ready                  := L      1.3,
           T_CHK1                   := T#20S,
           T_CHK2                   := T#20S,
           PB_Error_Rst             := L      1.5,
           M_FLICK                  := L      1.6,
           M_Adv_Err                := M   1620.4,
           M_Ret_Err                := M   1620.5,
           Visu_Adv                 := DB51.DBW  448,
           Visu_Ret                 := DB51.DBW  450);
      NOP   0;
NETWORK
TITLE =
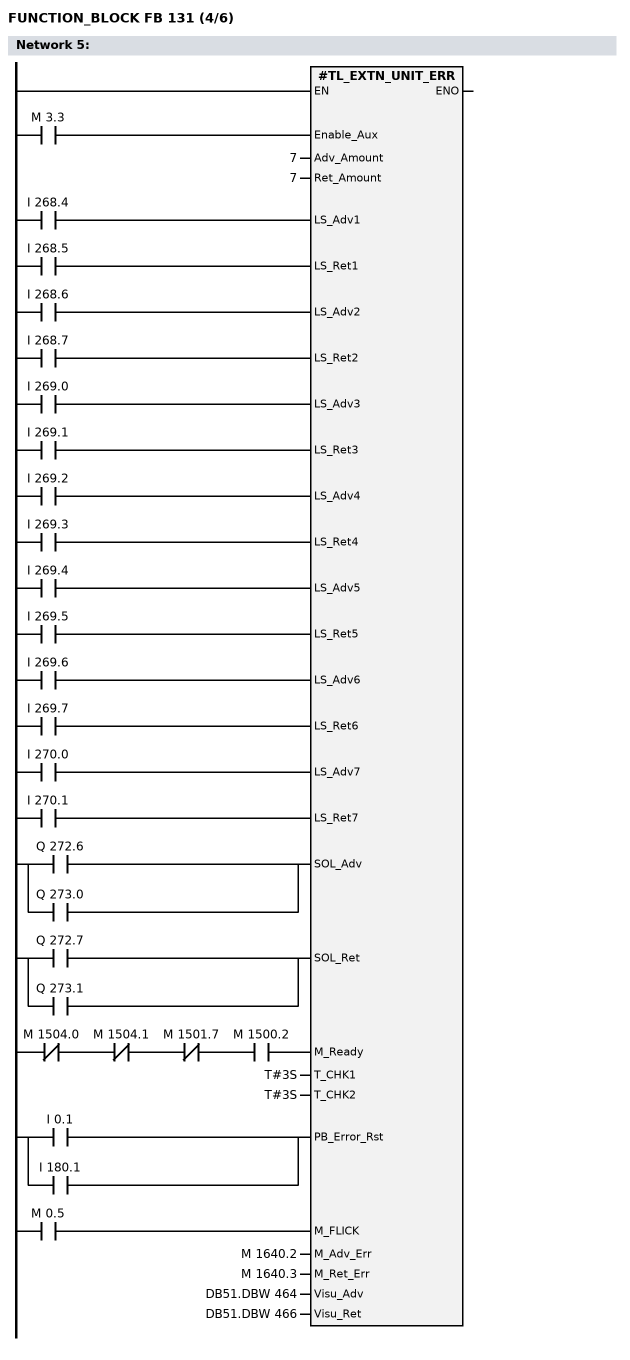

      A     M      3.3;
      =     L      0.0;
      BLD   103;
      A     I    268.4;
      =     L      0.1;
      BLD   103;
      A     I    268.5;
      =     L      0.2;
      BLD   103;
      A     I    268.6;
      =     L      0.3;
      BLD   103;
      A     I    268.7;
      =     L      0.4;
      BLD   103;
      A     I    269.0;
      =     L      0.5;
      BLD   103;
      A     I    269.1;
      =     L      0.6;
      BLD   103;
      A     I    269.2;
      =     L      0.7;
      BLD   103;
      A     I    269.3;
      =     L      1.0;
      BLD   103;
      A     I    269.4;
      =     L      1.1;
      BLD   103;
      A     I    269.5;
      =     L      1.2;
      BLD   103;
      A     I    269.6;
      =     L      1.3;
      BLD   103;
      A     I    269.7;
      =     L      1.4;
      BLD   103;
      A     I    270.0;
      =     L      1.5;
      BLD   103;
      A     I    270.1;
      =     L      1.6;
      BLD   103;
      A(    ;
      O     Q    272.6;
      O     Q    273.0;
      )     ;
      =     L      2.1;
      BLD   103;
      A(    ;
      O     Q    272.7;
      O     Q    273.1;
      )     ;
      =     L      2.2;
      BLD   103;
      AN    M   1504.0;
      AN    M   1504.1;
      AN    M   1501.7;
      A     M   1500.2;
      =     L      2.3;
      BLD   103;
      A(    ;
      O     I      0.1;
      O     I    180.1;
      )     ;
      =     L      2.5;
      BLD   103;
      A     M      0.5;
      =     L      2.6;
      BLD   103;
      CALL #TL_EXTN_UNIT_ERR (
           Enable_Aux               := L      0.0,
           Adv_Amount               := 7,
           Ret_Amount               := 7,
           LS_Adv1                  := L      0.1,
           LS_Ret1                  := L      0.2,
           LS_Adv2                  := L      0.3,
           LS_Ret2                  := L      0.4,
           LS_Adv3                  := L      0.5,
           LS_Ret3                  := L      0.6,
           LS_Adv4                  := L      0.7,
           LS_Ret4                  := L      1.0,
           LS_Adv5                  := L      1.1,
           LS_Ret5                  := L      1.2,
           LS_Adv6                  := L      1.3,
           LS_Ret6                  := L      1.4,
           LS_Adv7                  := L      1.5,
           LS_Ret7                  := L      1.6,
           SOL_Adv                  := L      2.1,
           SOL_Ret                  := L      2.2,
           M_Ready                  := L      2.3,
           T_CHK1                   := T#3S,
           T_CHK2                   := T#3S,
           PB_Error_Rst             := L      2.5,
           M_FLICK                  := L      2.6,
           M_Adv_Err                := M   1640.2,
           M_Ret_Err                := M   1640.3,
           Visu_Adv                 := DB51.DBW  464,
           Visu_Ret                 := DB51.DBW  466);
      NOP   0;
NETWORK
TITLE =
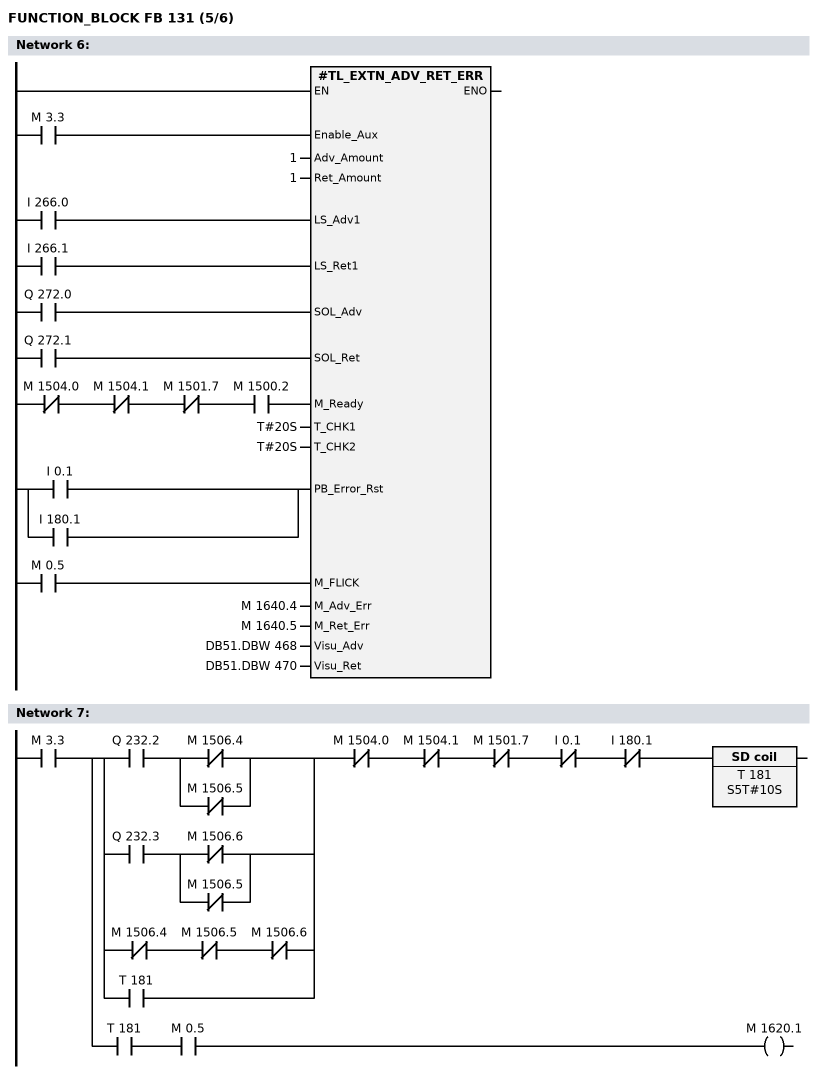

      A     M      3.3;
      =     L      0.0;
      BLD   103;
      A     I    266.0;
      =     L      0.1;
      BLD   103;
      A     I    266.1;
      =     L      0.2;
      BLD   103;
      A     Q    272.0;
      =     L      1.1;
      BLD   103;
      A     Q    272.1;
      =     L      1.2;
      BLD   103;
      AN    M   1504.0;
      AN    M   1504.1;
      AN    M   1501.7;
      A     M   1500.2;
      =     L      1.3;
      BLD   103;
      A(    ;
      O     I      0.1;
      O     I    180.1;
      )     ;
      =     L      1.5;
      BLD   103;
      A     M      0.5;
      =     L      1.6;
      BLD   103;
      CALL #TL_EXTN_ADV_RET_ERR (
           Enable_Aux               := L      0.0,
           Adv_Amount               := 1,
           Ret_Amount               := 1,
           LS_Adv1                  := L      0.1,
           LS_Ret1                  := L      0.2,
           SOL_Adv                  := L      1.1,
           SOL_Ret                  := L      1.2,
           M_Ready                  := L      1.3,
           T_CHK1                   := T#20S,
           T_CHK2                   := T#20S,
           PB_Error_Rst             := L      1.5,
           M_FLICK                  := L      1.6,
           M_Adv_Err                := M   1640.4,
           M_Ret_Err                := M   1640.5,
           Visu_Adv                 := DB51.DBW  468,
           Visu_Ret                 := DB51.DBW  470);
      NOP   0;
NETWORK
TITLE =

      A     M      3.3;
      =     L      0.0;
      A     L      0.0;
      A(    ;
      A     Q    232.2;
      A(    ;
      ON    M   1506.4;
      ON    M   1506.5;
      )     ;
      O     ;
      A     Q    232.3;
      A(    ;
      ON    M   1506.6;
      ON    M   1506.5;
      )     ;
      O     ;
      AN    M   1506.4;
      AN    M   1506.5;
      AN    M   1506.6;
      O     T    181;
      )     ;
      AN    M   1504.0;
      AN    M   1504.1;
      AN    M   1501.7;
      AN    I      0.1;
      AN    I    180.1;
      L     S5T#10S;
      SD    T    181;
      A     L      0.0;
      A     T    181;
      A     M      0.5;
      =     M   1620.1;
NETWORK
TITLE =
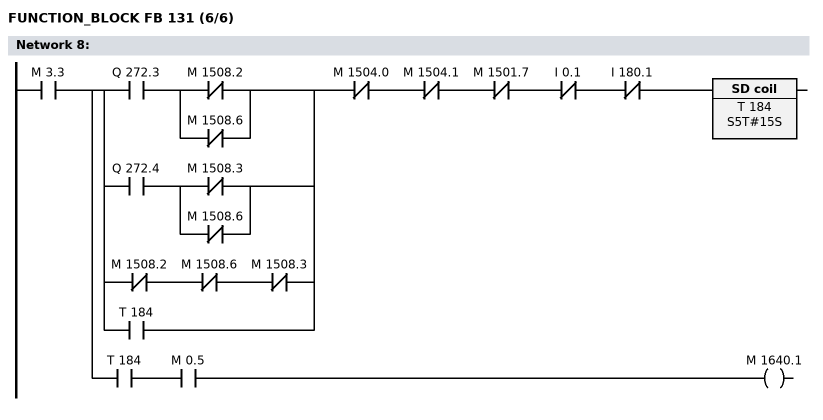

      A     M      3.3;
      =     L      0.0;
      A     L      0.0;
      A(    ;
      A     Q    272.3;
      A(    ;
      ON    M   1508.2;
      ON    M   1508.6;
      )     ;
      O     ;
      A     Q    272.4;
      A(    ;
      ON    M   1508.3;
      ON    M   1508.6;
      )     ;
      O     ;
      AN    M   1508.2;
      AN    M   1508.6;
      AN    M   1508.3;
      O     T    184;
      )     ;
      AN    M   1504.0;
      AN    M   1504.1;
      AN    M   1501.7;
      AN    I      0.1;
      AN    I    180.1;
      L     S5T#15S;
      SD    T    184;
      A     L      0.0;
      A     T    184;
      A     M      0.5;
      =     M   1640.1;
END_FUNCTION_BLOCK

DATA_BLOCK DB 131
TITLE =
VERSION : 0.0

 FB 131
BEGIN
   S701_FDR_A_STORAGE_ERR.Enable_Aux := FALSE;
   S701_FDR_A_STORAGE_ERR.Adv_Amount := 0;
   S701_FDR_A_STORAGE_ERR.Ret_Amount := 0;
   S701_FDR_A_STORAGE_ERR.LS_Adv1 := FALSE;
   S701_FDR_A_STORAGE_ERR.LS_Ret1 := FALSE;
   S701_FDR_A_STORAGE_ERR.LS_Adv2 := FALSE;
   S701_FDR_A_STORAGE_ERR.LS_Ret2 := FALSE;
   S701_FDR_A_STORAGE_ERR.LS_Adv3 := FALSE;
   S701_FDR_A_STORAGE_ERR.LS_Ret3 := FALSE;
   S701_FDR_A_STORAGE_ERR.LS_Adv4 := FALSE;
   S701_FDR_A_STORAGE_ERR.LS_Ret4 := FALSE;
   S701_FDR_A_STORAGE_ERR.SOL_Adv := FALSE;
   S701_FDR_A_STORAGE_ERR.SOL_Ret := FALSE;
   S701_FDR_A_STORAGE_ERR.M_Ready := FALSE;
   S701_FDR_A_STORAGE_ERR.T_CHK1 := T#0MS;
   S701_FDR_A_STORAGE_ERR.T_CHK2 := T#0MS;
   S701_FDR_A_STORAGE_ERR.PB_Lamp_CHK := FALSE;
   S701_FDR_A_STORAGE_ERR.PB_Error_Rst := FALSE;
   S701_FDR_A_STORAGE_ERR.M_FLICK := FALSE;
   S701_FDR_A_STORAGE_ERR.M_Adv_Err := FALSE;
   S701_FDR_A_STORAGE_ERR.M_Ret_Err := FALSE;
   S701_FDR_A_STORAGE_ERR.LP_Adv := FALSE;
   S701_FDR_A_STORAGE_ERR.LP_Ret := FALSE;
   S701_FDR_A_STORAGE_ERR.Visu_Adv := W#16#0;
   S701_FDR_A_STORAGE_ERR.Visu_Ret := W#16#0;
   S701_FDR_A_STORAGE_ERR.Error_T1.IN := FALSE;
   S701_FDR_A_STORAGE_ERR.Error_T1.PT := T#0MS;
   S701_FDR_A_STORAGE_ERR.Error_T1.Q := FALSE;
   S701_FDR_A_STORAGE_ERR.Error_T1.ET := T#0MS;
   S701_FDR_A_STORAGE_ERR.Error_T1.STATE := B#16#0;
   S701_FDR_A_STORAGE_ERR.Error_T1.STIME := T#0MS;
   S701_FDR_A_STORAGE_ERR.Error_T1.ATIME := T#0MS;
   S701_FDR_A_STORAGE_ERR.Error_T2.IN := FALSE;
   S701_FDR_A_STORAGE_ERR.Error_T2.PT := T#0MS;
   S701_FDR_A_STORAGE_ERR.Error_T2.Q := FALSE;
   S701_FDR_A_STORAGE_ERR.Error_T2.ET := T#0MS;
   S701_FDR_A_STORAGE_ERR.Error_T2.STATE := B#16#0;
   S701_FDR_A_STORAGE_ERR.Error_T2.STIME := T#0MS;
   S701_FDR_A_STORAGE_ERR.Error_T2.ATIME := T#0MS;
   S701_FDR_A_STORAGE_ERR.CHK_Aux1 := FALSE;
   S701_FDR_A_STORAGE_ERR.CHK_Aux2 := FALSE;
   S701_FDR_A_STORAGE_ERR.Error_T1_DN := FALSE;
   S701_FDR_A_STORAGE_ERR.Error_T2_DN := FALSE;
   S701_FDR_A_STORAGE_ERR.Adv_Memo := FALSE;
   S701_FDR_A_STORAGE_ERR.Visu_Adv_Arr[0] := FALSE;
   S701_FDR_A_STORAGE_ERR.Visu_Adv_Arr[1] := FALSE;
   S701_FDR_A_STORAGE_ERR.Visu_Adv_Arr[2] := FALSE;
   S701_FDR_A_STORAGE_ERR.Visu_Adv_Arr[3] := FALSE;
   S701_FDR_A_STORAGE_ERR.Visu_Adv_Arr[4] := FALSE;
   S701_FDR_A_STORAGE_ERR.Visu_Adv_Arr[5] := FALSE;
   S701_FDR_A_STORAGE_ERR.Visu_Adv_Arr[6] := FALSE;
   S701_FDR_A_STORAGE_ERR.Visu_Adv_Arr[7] := FALSE;
   S701_FDR_A_STORAGE_ERR.Visu_Adv_Arr[8] := FALSE;
   S701_FDR_A_STORAGE_ERR.Visu_Adv_Arr[9] := FALSE;
   S701_FDR_A_STORAGE_ERR.Visu_Adv_Arr[10] := FALSE;
   S701_FDR_A_STORAGE_ERR.Visu_Adv_Arr[11] := FALSE;
   S701_FDR_A_STORAGE_ERR.Visu_Adv_Arr[12] := FALSE;
   S701_FDR_A_STORAGE_ERR.Visu_Adv_Arr[13] := FALSE;
   S701_FDR_A_STORAGE_ERR.Visu_Adv_Arr[14] := FALSE;
   S701_FDR_A_STORAGE_ERR.Visu_Adv_Arr[15] := FALSE;
   S701_FDR_A_STORAGE_ERR.Visu_Ret_Arr[0] := FALSE;
   S701_FDR_A_STORAGE_ERR.Visu_Ret_Arr[1] := FALSE;
   S701_FDR_A_STORAGE_ERR.Visu_Ret_Arr[2] := FALSE;
   S701_FDR_A_STORAGE_ERR.Visu_Ret_Arr[3] := FALSE;
   S701_FDR_A_STORAGE_ERR.Visu_Ret_Arr[4] := FALSE;
   S701_FDR_A_STORAGE_ERR.Visu_Ret_Arr[5] := FALSE;
   S701_FDR_A_STORAGE_ERR.Visu_Ret_Arr[6] := FALSE;
   S701_FDR_A_STORAGE_ERR.Visu_Ret_Arr[7] := FALSE;
   S701_FDR_A_STORAGE_ERR.Visu_Ret_Arr[8] := FALSE;
   S701_FDR_A_STORAGE_ERR.Visu_Ret_Arr[9] := FALSE;
   S701_FDR_A_STORAGE_ERR.Visu_Ret_Arr[10] := FALSE;
   S701_FDR_A_STORAGE_ERR.Visu_Ret_Arr[11] := FALSE;
   S701_FDR_A_STORAGE_ERR.Visu_Ret_Arr[12] := FALSE;
   S701_FDR_A_STORAGE_ERR.Visu_Ret_Arr[13] := FALSE;
   S701_FDR_A_STORAGE_ERR.Visu_Ret_Arr[14] := FALSE;
   S701_FDR_A_STORAGE_ERR.Visu_Ret_Arr[15] := FALSE;
   S701_FDR_A_STORAGE_ERR.BLK_Move_Ret := 0;
   S701_FDR_A_STORAGE_ERR.Enable := FALSE;
   S701_FDR_A_STORAGE_ERR.Adv_End := FALSE;
   S701_FDR_A_STORAGE_ERR.Ret_End := FALSE;
   S701_FDR_B_STORAGE_ERR.Enable_Aux := FALSE;
   S701_FDR_B_STORAGE_ERR.Adv_Amount := 0;
   S701_FDR_B_STORAGE_ERR.Ret_Amount := 0;
   S701_FDR_B_STORAGE_ERR.LS_Adv1 := FALSE;
   S701_FDR_B_STORAGE_ERR.LS_Ret1 := FALSE;
   S701_FDR_B_STORAGE_ERR.LS_Adv2 := FALSE;
   S701_FDR_B_STORAGE_ERR.LS_Ret2 := FALSE;
   S701_FDR_B_STORAGE_ERR.LS_Adv3 := FALSE;
   S701_FDR_B_STORAGE_ERR.LS_Ret3 := FALSE;
   S701_FDR_B_STORAGE_ERR.LS_Adv4 := FALSE;
   S701_FDR_B_STORAGE_ERR.LS_Ret4 := FALSE;
   S701_FDR_B_STORAGE_ERR.SOL_Adv := FALSE;
   S701_FDR_B_STORAGE_ERR.SOL_Ret := FALSE;
   S701_FDR_B_STORAGE_ERR.M_Ready := FALSE;
   S701_FDR_B_STORAGE_ERR.T_CHK1 := T#0MS;
   S701_FDR_B_STORAGE_ERR.T_CHK2 := T#0MS;
   S701_FDR_B_STORAGE_ERR.PB_Lamp_CHK := FALSE;
   S701_FDR_B_STORAGE_ERR.PB_Error_Rst := FALSE;
   S701_FDR_B_STORAGE_ERR.M_FLICK := FALSE;
   S701_FDR_B_STORAGE_ERR.M_Adv_Err := FALSE;
   S701_FDR_B_STORAGE_ERR.M_Ret_Err := FALSE;
   S701_FDR_B_STORAGE_ERR.LP_Adv := FALSE;
   S701_FDR_B_STORAGE_ERR.LP_Ret := FALSE;
   S701_FDR_B_STORAGE_ERR.Visu_Adv := W#16#0;
   S701_FDR_B_STORAGE_ERR.Visu_Ret := W#16#0;
   S701_FDR_B_STORAGE_ERR.Error_T1.IN := FALSE;
   S701_FDR_B_STORAGE_ERR.Error_T1.PT := T#0MS;
   S701_FDR_B_STORAGE_ERR.Error_T1.Q := FALSE;
   S701_FDR_B_STORAGE_ERR.Error_T1.ET := T#0MS;
   S701_FDR_B_STORAGE_ERR.Error_T1.STATE := B#16#0;
   S701_FDR_B_STORAGE_ERR.Error_T1.STIME := T#0MS;
   S701_FDR_B_STORAGE_ERR.Error_T1.ATIME := T#0MS;
   S701_FDR_B_STORAGE_ERR.Error_T2.IN := FALSE;
   S701_FDR_B_STORAGE_ERR.Error_T2.PT := T#0MS;
   S701_FDR_B_STORAGE_ERR.Error_T2.Q := FALSE;
   S701_FDR_B_STORAGE_ERR.Error_T2.ET := T#0MS;
   S701_FDR_B_STORAGE_ERR.Error_T2.STATE := B#16#0;
   S701_FDR_B_STORAGE_ERR.Error_T2.STIME := T#0MS;
   S701_FDR_B_STORAGE_ERR.Error_T2.ATIME := T#0MS;
   S701_FDR_B_STORAGE_ERR.CHK_Aux1 := FALSE;
   S701_FDR_B_STORAGE_ERR.CHK_Aux2 := FALSE;
   S701_FDR_B_STORAGE_ERR.Error_T1_DN := FALSE;
   S701_FDR_B_STORAGE_ERR.Error_T2_DN := FALSE;
   S701_FDR_B_STORAGE_ERR.Adv_Memo := FALSE;
   S701_FDR_B_STORAGE_ERR.Visu_Adv_Arr[0] := FALSE;
   S701_FDR_B_STORAGE_ERR.Visu_Adv_Arr[1] := FALSE;
   S701_FDR_B_STORAGE_ERR.Visu_Adv_Arr[2] := FALSE;
   S701_FDR_B_STORAGE_ERR.Visu_Adv_Arr[3] := FALSE;
   S701_FDR_B_STORAGE_ERR.Visu_Adv_Arr[4] := FALSE;
   S701_FDR_B_STORAGE_ERR.Visu_Adv_Arr[5] := FALSE;
   S701_FDR_B_STORAGE_ERR.Visu_Adv_Arr[6] := FALSE;
   S701_FDR_B_STORAGE_ERR.Visu_Adv_Arr[7] := FALSE;
   S701_FDR_B_STORAGE_ERR.Visu_Adv_Arr[8] := FALSE;
   S701_FDR_B_STORAGE_ERR.Visu_Adv_Arr[9] := FALSE;
   S701_FDR_B_STORAGE_ERR.Visu_Adv_Arr[10] := FALSE;
   S701_FDR_B_STORAGE_ERR.Visu_Adv_Arr[11] := FALSE;
   S701_FDR_B_STORAGE_ERR.Visu_Adv_Arr[12] := FALSE;
   S701_FDR_B_STORAGE_ERR.Visu_Adv_Arr[13] := FALSE;
   S701_FDR_B_STORAGE_ERR.Visu_Adv_Arr[14] := FALSE;
   S701_FDR_B_STORAGE_ERR.Visu_Adv_Arr[15] := FALSE;
   S701_FDR_B_STORAGE_ERR.Visu_Ret_Arr[0] := FALSE;
   S701_FDR_B_STORAGE_ERR.Visu_Ret_Arr[1] := FALSE;
   S701_FDR_B_STORAGE_ERR.Visu_Ret_Arr[2] := FALSE;
   S701_FDR_B_STORAGE_ERR.Visu_Ret_Arr[3] := FALSE;
   S701_FDR_B_STORAGE_ERR.Visu_Ret_Arr[4] := FALSE;
   S701_FDR_B_STORAGE_ERR.Visu_Ret_Arr[5] := FALSE;
   S701_FDR_B_STORAGE_ERR.Visu_Ret_Arr[6] := FALSE;
   S701_FDR_B_STORAGE_ERR.Visu_Ret_Arr[7] := FALSE;
   S701_FDR_B_STORAGE_ERR.Visu_Ret_Arr[8] := FALSE;
   S701_FDR_B_STORAGE_ERR.Visu_Ret_Arr[9] := FALSE;
   S701_FDR_B_STORAGE_ERR.Visu_Ret_Arr[10] := FALSE;
   S701_FDR_B_STORAGE_ERR.Visu_Ret_Arr[11] := FALSE;
   S701_FDR_B_STORAGE_ERR.Visu_Ret_Arr[12] := FALSE;
   S701_FDR_B_STORAGE_ERR.Visu_Ret_Arr[13] := FALSE;
   S701_FDR_B_STORAGE_ERR.Visu_Ret_Arr[14] := FALSE;
   S701_FDR_B_STORAGE_ERR.Visu_Ret_Arr[15] := FALSE;
   S701_FDR_B_STORAGE_ERR.BLK_Move_Ret := 0;
   S701_FDR_B_STORAGE_ERR.Enable := FALSE;
   S701_FDR_B_STORAGE_ERR.Adv_End := FALSE;
   S701_FDR_B_STORAGE_ERR.Ret_End := FALSE;
   LM_EXTN_UNIT_ERR.Enable_Aux := FALSE;
   LM_EXTN_UNIT_ERR.Adv_Amount := 0;
   LM_EXTN_UNIT_ERR.Ret_Amount := 0;
   LM_EXTN_UNIT_ERR.LS_Adv1 := FALSE;
   LM_EXTN_UNIT_ERR.LS_Ret1 := FALSE;
   LM_EXTN_UNIT_ERR.LS_Adv2 := FALSE;
   LM_EXTN_UNIT_ERR.LS_Ret2 := FALSE;
   LM_EXTN_UNIT_ERR.LS_Adv3 := FALSE;
   LM_EXTN_UNIT_ERR.LS_Ret3 := FALSE;
   LM_EXTN_UNIT_ERR.LS_Adv4 := FALSE;
   LM_EXTN_UNIT_ERR.LS_Ret4 := FALSE;
   LM_EXTN_UNIT_ERR.LS_Adv5 := FALSE;
   LM_EXTN_UNIT_ERR.LS_Ret5 := FALSE;
   LM_EXTN_UNIT_ERR.LS_Adv6 := FALSE;
   LM_EXTN_UNIT_ERR.LS_Ret6 := FALSE;
   LM_EXTN_UNIT_ERR.LS_Adv7 := FALSE;
   LM_EXTN_UNIT_ERR.LS_Ret7 := FALSE;
   LM_EXTN_UNIT_ERR.LS_Adv8 := FALSE;
   LM_EXTN_UNIT_ERR.LS_Ret8 := FALSE;
   LM_EXTN_UNIT_ERR.SOL_Adv := FALSE;
   LM_EXTN_UNIT_ERR.SOL_Ret := FALSE;
   LM_EXTN_UNIT_ERR.M_Ready := FALSE;
   LM_EXTN_UNIT_ERR.T_CHK1 := T#0MS;
   LM_EXTN_UNIT_ERR.T_CHK2 := T#0MS;
   LM_EXTN_UNIT_ERR.PB_Lamp_CHK := FALSE;
   LM_EXTN_UNIT_ERR.PB_Error_Rst := FALSE;
   LM_EXTN_UNIT_ERR.M_FLICK := FALSE;
   LM_EXTN_UNIT_ERR.M_Adv_Err := FALSE;
   LM_EXTN_UNIT_ERR.M_Ret_Err := FALSE;
   LM_EXTN_UNIT_ERR.LP_Adv := FALSE;
   LM_EXTN_UNIT_ERR.LP_Ret := FALSE;
   LM_EXTN_UNIT_ERR.Visu_Adv := W#16#0;
   LM_EXTN_UNIT_ERR.Visu_Ret := W#16#0;
   LM_EXTN_UNIT_ERR.Error_T1.IN := FALSE;
   LM_EXTN_UNIT_ERR.Error_T1.PT := T#0MS;
   LM_EXTN_UNIT_ERR.Error_T1.Q := FALSE;
   LM_EXTN_UNIT_ERR.Error_T1.ET := T#0MS;
   LM_EXTN_UNIT_ERR.Error_T1.STATE := B#16#0;
   LM_EXTN_UNIT_ERR.Error_T1.STIME := T#0MS;
   LM_EXTN_UNIT_ERR.Error_T1.ATIME := T#0MS;
   LM_EXTN_UNIT_ERR.Error_T2.IN := FALSE;
   LM_EXTN_UNIT_ERR.Error_T2.PT := T#0MS;
   LM_EXTN_UNIT_ERR.Error_T2.Q := FALSE;
   LM_EXTN_UNIT_ERR.Error_T2.ET := T#0MS;
   LM_EXTN_UNIT_ERR.Error_T2.STATE := B#16#0;
   LM_EXTN_UNIT_ERR.Error_T2.STIME := T#0MS;
   LM_EXTN_UNIT_ERR.Error_T2.ATIME := T#0MS;
   LM_EXTN_UNIT_ERR.Adv_End_Aux := FALSE;
   LM_EXTN_UNIT_ERR.Ret_End_Aux := FALSE;
   LM_EXTN_UNIT_ERR.CHK_Aux1 := FALSE;
   LM_EXTN_UNIT_ERR.CHK_Aux2 := FALSE;
   LM_EXTN_UNIT_ERR.Error_T1_DN := FALSE;
   LM_EXTN_UNIT_ERR.Error_T2_DN := FALSE;
   LM_EXTN_UNIT_ERR.Adv_Memo := FALSE;
   LM_EXTN_UNIT_ERR.Visu_Adv_Arr[0] := FALSE;
   LM_EXTN_UNIT_ERR.Visu_Adv_Arr[1] := FALSE;
   LM_EXTN_UNIT_ERR.Visu_Adv_Arr[2] := FALSE;
   LM_EXTN_UNIT_ERR.Visu_Adv_Arr[3] := FALSE;
   LM_EXTN_UNIT_ERR.Visu_Adv_Arr[4] := FALSE;
   LM_EXTN_UNIT_ERR.Visu_Adv_Arr[5] := FALSE;
   LM_EXTN_UNIT_ERR.Visu_Adv_Arr[6] := FALSE;
   LM_EXTN_UNIT_ERR.Visu_Adv_Arr[7] := FALSE;
   LM_EXTN_UNIT_ERR.Visu_Adv_Arr[8] := FALSE;
   LM_EXTN_UNIT_ERR.Visu_Adv_Arr[9] := FALSE;
   LM_EXTN_UNIT_ERR.Visu_Adv_Arr[10] := FALSE;
   LM_EXTN_UNIT_ERR.Visu_Adv_Arr[11] := FALSE;
   LM_EXTN_UNIT_ERR.Visu_Adv_Arr[12] := FALSE;
   LM_EXTN_UNIT_ERR.Visu_Adv_Arr[13] := FALSE;
   LM_EXTN_UNIT_ERR.Visu_Adv_Arr[14] := FALSE;
   LM_EXTN_UNIT_ERR.Visu_Adv_Arr[15] := FALSE;
   LM_EXTN_UNIT_ERR.Visu_Ret_Arr[0] := FALSE;
   LM_EXTN_UNIT_ERR.Visu_Ret_Arr[1] := FALSE;
   LM_EXTN_UNIT_ERR.Visu_Ret_Arr[2] := FALSE;
   LM_EXTN_UNIT_ERR.Visu_Ret_Arr[3] := FALSE;
   LM_EXTN_UNIT_ERR.Visu_Ret_Arr[4] := FALSE;
   LM_EXTN_UNIT_ERR.Visu_Ret_Arr[5] := FALSE;
   LM_EXTN_UNIT_ERR.Visu_Ret_Arr[6] := FALSE;
   LM_EXTN_UNIT_ERR.Visu_Ret_Arr[7] := FALSE;
   LM_EXTN_UNIT_ERR.Visu_Ret_Arr[8] := FALSE;
   LM_EXTN_UNIT_ERR.Visu_Ret_Arr[9] := FALSE;
   LM_EXTN_UNIT_ERR.Visu_Ret_Arr[10] := FALSE;
   LM_EXTN_UNIT_ERR.Visu_Ret_Arr[11] := FALSE;
   LM_EXTN_UNIT_ERR.Visu_Ret_Arr[12] := FALSE;
   LM_EXTN_UNIT_ERR.Visu_Ret_Arr[13] := FALSE;
   LM_EXTN_UNIT_ERR.Visu_Ret_Arr[14] := FALSE;
   LM_EXTN_UNIT_ERR.Visu_Ret_Arr[15] := FALSE;
   LM_EXTN_UNIT_ERR.BLK_Move_Ret := 0;
   LM_EXTN_UNIT_ERR.Enable := FALSE;
   LM_EXTN_UNIT_ERR.Adv_End := FALSE;
   LM_EXTN_UNIT_ERR.Ret_End := FALSE;
   LM_EXTN_ADV_RET_ERR.Enable_Aux := FALSE;
   LM_EXTN_ADV_RET_ERR.Adv_Amount := 0;
   LM_EXTN_ADV_RET_ERR.Ret_Amount := 0;
   LM_EXTN_ADV_RET_ERR.LS_Adv1 := FALSE;
   LM_EXTN_ADV_RET_ERR.LS_Ret1 := FALSE;
   LM_EXTN_ADV_RET_ERR.LS_Adv2 := FALSE;
   LM_EXTN_ADV_RET_ERR.LS_Ret2 := FALSE;
   LM_EXTN_ADV_RET_ERR.LS_Adv3 := FALSE;
   LM_EXTN_ADV_RET_ERR.LS_Ret3 := FALSE;
   LM_EXTN_ADV_RET_ERR.LS_Adv4 := FALSE;
   LM_EXTN_ADV_RET_ERR.LS_Ret4 := FALSE;
   LM_EXTN_ADV_RET_ERR.SOL_Adv := FALSE;
   LM_EXTN_ADV_RET_ERR.SOL_Ret := FALSE;
   LM_EXTN_ADV_RET_ERR.M_Ready := FALSE;
   LM_EXTN_ADV_RET_ERR.T_CHK1 := T#0MS;
   LM_EXTN_ADV_RET_ERR.T_CHK2 := T#0MS;
   LM_EXTN_ADV_RET_ERR.PB_Lamp_CHK := FALSE;
   LM_EXTN_ADV_RET_ERR.PB_Error_Rst := FALSE;
   LM_EXTN_ADV_RET_ERR.M_FLICK := FALSE;
   LM_EXTN_ADV_RET_ERR.M_Adv_Err := FALSE;
   LM_EXTN_ADV_RET_ERR.M_Ret_Err := FALSE;
   LM_EXTN_ADV_RET_ERR.LP_Adv := FALSE;
   LM_EXTN_ADV_RET_ERR.LP_Ret := FALSE;
   LM_EXTN_ADV_RET_ERR.Visu_Adv := W#16#0;
   LM_EXTN_ADV_RET_ERR.Visu_Ret := W#16#0;
   LM_EXTN_ADV_RET_ERR.Error_T1.IN := FALSE;
   LM_EXTN_ADV_RET_ERR.Error_T1.PT := T#0MS;
   LM_EXTN_ADV_RET_ERR.Error_T1.Q := FALSE;
   LM_EXTN_ADV_RET_ERR.Error_T1.ET := T#0MS;
   LM_EXTN_ADV_RET_ERR.Error_T1.STATE := B#16#0;
   LM_EXTN_ADV_RET_ERR.Error_T1.STIME := T#0MS;
   LM_EXTN_ADV_RET_ERR.Error_T1.ATIME := T#0MS;
   LM_EXTN_ADV_RET_ERR.Error_T2.IN := FALSE;
   LM_EXTN_ADV_RET_ERR.Error_T2.PT := T#0MS;
   LM_EXTN_ADV_RET_ERR.Error_T2.Q := FALSE;
   LM_EXTN_ADV_RET_ERR.Error_T2.ET := T#0MS;
   LM_EXTN_ADV_RET_ERR.Error_T2.STATE := B#16#0;
   LM_EXTN_ADV_RET_ERR.Error_T2.STIME := T#0MS;
   LM_EXTN_ADV_RET_ERR.Error_T2.ATIME := T#0MS;
   LM_EXTN_ADV_RET_ERR.CHK_Aux1 := FALSE;
   LM_EXTN_ADV_RET_ERR.CHK_Aux2 := FALSE;
   LM_EXTN_ADV_RET_ERR.Error_T1_DN := FALSE;
   LM_EXTN_ADV_RET_ERR.Error_T2_DN := FALSE;
   LM_EXTN_ADV_RET_ERR.Adv_Memo := FALSE;
   LM_EXTN_ADV_RET_ERR.Visu_Adv_Arr[0] := FALSE;
   LM_EXTN_ADV_RET_ERR.Visu_Adv_Arr[1] := FALSE;
   LM_EXTN_ADV_RET_ERR.Visu_Adv_Arr[2] := FALSE;
   LM_EXTN_ADV_RET_ERR.Visu_Adv_Arr[3] := FALSE;
   LM_EXTN_ADV_RET_ERR.Visu_Adv_Arr[4] := FALSE;
   LM_EXTN_ADV_RET_ERR.Visu_Adv_Arr[5] := FALSE;
   LM_EXTN_ADV_RET_ERR.Visu_Adv_Arr[6] := FALSE;
   LM_EXTN_ADV_RET_ERR.Visu_Adv_Arr[7] := FALSE;
   LM_EXTN_ADV_RET_ERR.Visu_Adv_Arr[8] := FALSE;
   LM_EXTN_ADV_RET_ERR.Visu_Adv_Arr[9] := FALSE;
   LM_EXTN_ADV_RET_ERR.Visu_Adv_Arr[10] := FALSE;
   LM_EXTN_ADV_RET_ERR.Visu_Adv_Arr[11] := FALSE;
   LM_EXTN_ADV_RET_ERR.Visu_Adv_Arr[12] := FALSE;
   LM_EXTN_ADV_RET_ERR.Visu_Adv_Arr[13] := FALSE;
   LM_EXTN_ADV_RET_ERR.Visu_Adv_Arr[14] := FALSE;
   LM_EXTN_ADV_RET_ERR.Visu_Adv_Arr[15] := FALSE;
   LM_EXTN_ADV_RET_ERR.Visu_Ret_Arr[0] := FALSE;
   LM_EXTN_ADV_RET_ERR.Visu_Ret_Arr[1] := FALSE;
   LM_EXTN_ADV_RET_ERR.Visu_Ret_Arr[2] := FALSE;
   LM_EXTN_ADV_RET_ERR.Visu_Ret_Arr[3] := FALSE;
   LM_EXTN_ADV_RET_ERR.Visu_Ret_Arr[4] := FALSE;
   LM_EXTN_ADV_RET_ERR.Visu_Ret_Arr[5] := FALSE;
   LM_EXTN_ADV_RET_ERR.Visu_Ret_Arr[6] := FALSE;
   LM_EXTN_ADV_RET_ERR.Visu_Ret_Arr[7] := FALSE;
   LM_EXTN_ADV_RET_ERR.Visu_Ret_Arr[8] := FALSE;
   LM_EXTN_ADV_RET_ERR.Visu_Ret_Arr[9] := FALSE;
   LM_EXTN_ADV_RET_ERR.Visu_Ret_Arr[10] := FALSE;
   LM_EXTN_ADV_RET_ERR.Visu_Ret_Arr[11] := FALSE;
   LM_EXTN_ADV_RET_ERR.Visu_Ret_Arr[12] := FALSE;
   LM_EXTN_ADV_RET_ERR.Visu_Ret_Arr[13] := FALSE;
   LM_EXTN_ADV_RET_ERR.Visu_Ret_Arr[14] := FALSE;
   LM_EXTN_ADV_RET_ERR.Visu_Ret_Arr[15] := FALSE;
   LM_EXTN_ADV_RET_ERR.BLK_Move_Ret := 0;
   LM_EXTN_ADV_RET_ERR.Enable := FALSE;
   LM_EXTN_ADV_RET_ERR.Adv_End := FALSE;
   LM_EXTN_ADV_RET_ERR.Ret_End := FALSE;
   TL_EXTN_UNIT_ERR.Enable_Aux := FALSE;
   TL_EXTN_UNIT_ERR.Adv_Amount := 0;
   TL_EXTN_UNIT_ERR.Ret_Amount := 0;
   TL_EXTN_UNIT_ERR.LS_Adv1 := FALSE;
   TL_EXTN_UNIT_ERR.LS_Ret1 := FALSE;
   TL_EXTN_UNIT_ERR.LS_Adv2 := FALSE;
   TL_EXTN_UNIT_ERR.LS_Ret2 := FALSE;
   TL_EXTN_UNIT_ERR.LS_Adv3 := FALSE;
   TL_EXTN_UNIT_ERR.LS_Ret3 := FALSE;
   TL_EXTN_UNIT_ERR.LS_Adv4 := FALSE;
   TL_EXTN_UNIT_ERR.LS_Ret4 := FALSE;
   TL_EXTN_UNIT_ERR.LS_Adv5 := FALSE;
   TL_EXTN_UNIT_ERR.LS_Ret5 := FALSE;
   TL_EXTN_UNIT_ERR.LS_Adv6 := FALSE;
   TL_EXTN_UNIT_ERR.LS_Ret6 := FALSE;
   TL_EXTN_UNIT_ERR.LS_Adv7 := FALSE;
   TL_EXTN_UNIT_ERR.LS_Ret7 := FALSE;
   TL_EXTN_UNIT_ERR.LS_Adv8 := FALSE;
   TL_EXTN_UNIT_ERR.LS_Ret8 := FALSE;
   TL_EXTN_UNIT_ERR.SOL_Adv := FALSE;
   TL_EXTN_UNIT_ERR.SOL_Ret := FALSE;
   TL_EXTN_UNIT_ERR.M_Ready := FALSE;
   TL_EXTN_UNIT_ERR.T_CHK1 := T#0MS;
   TL_EXTN_UNIT_ERR.T_CHK2 := T#0MS;
   TL_EXTN_UNIT_ERR.PB_Lamp_CHK := FALSE;
   TL_EXTN_UNIT_ERR.PB_Error_Rst := FALSE;
   TL_EXTN_UNIT_ERR.M_FLICK := FALSE;
   TL_EXTN_UNIT_ERR.M_Adv_Err := FALSE;
   TL_EXTN_UNIT_ERR.M_Ret_Err := FALSE;
   TL_EXTN_UNIT_ERR.LP_Adv := FALSE;
   TL_EXTN_UNIT_ERR.LP_Ret := FALSE;
   TL_EXTN_UNIT_ERR.Visu_Adv := W#16#0;
   TL_EXTN_UNIT_ERR.Visu_Ret := W#16#0;
   TL_EXTN_UNIT_ERR.Error_T1.IN := FALSE;
   TL_EXTN_UNIT_ERR.Error_T1.PT := T#0MS;
   TL_EXTN_UNIT_ERR.Error_T1.Q := FALSE;
   TL_EXTN_UNIT_ERR.Error_T1.ET := T#0MS;
   TL_EXTN_UNIT_ERR.Error_T1.STATE := B#16#0;
   TL_EXTN_UNIT_ERR.Error_T1.STIME := T#0MS;
   TL_EXTN_UNIT_ERR.Error_T1.ATIME := T#0MS;
   TL_EXTN_UNIT_ERR.Error_T2.IN := FALSE;
   TL_EXTN_UNIT_ERR.Error_T2.PT := T#0MS;
   TL_EXTN_UNIT_ERR.Error_T2.Q := FALSE;
   TL_EXTN_UNIT_ERR.Error_T2.ET := T#0MS;
   TL_EXTN_UNIT_ERR.Error_T2.STATE := B#16#0;
   TL_EXTN_UNIT_ERR.Error_T2.STIME := T#0MS;
   TL_EXTN_UNIT_ERR.Error_T2.ATIME := T#0MS;
   TL_EXTN_UNIT_ERR.Adv_End_Aux := FALSE;
   TL_EXTN_UNIT_ERR.Ret_End_Aux := FALSE;
   TL_EXTN_UNIT_ERR.CHK_Aux1 := FALSE;
   TL_EXTN_UNIT_ERR.CHK_Aux2 := FALSE;
   TL_EXTN_UNIT_ERR.Error_T1_DN := FALSE;
   TL_EXTN_UNIT_ERR.Error_T2_DN := FALSE;
   TL_EXTN_UNIT_ERR.Adv_Memo := FALSE;
   TL_EXTN_UNIT_ERR.Visu_Adv_Arr[0] := FALSE;
   TL_EXTN_UNIT_ERR.Visu_Adv_Arr[1] := FALSE;
   TL_EXTN_UNIT_ERR.Visu_Adv_Arr[2] := FALSE;
   TL_EXTN_UNIT_ERR.Visu_Adv_Arr[3] := FALSE;
   TL_EXTN_UNIT_ERR.Visu_Adv_Arr[4] := FALSE;
   TL_EXTN_UNIT_ERR.Visu_Adv_Arr[5] := FALSE;
   TL_EXTN_UNIT_ERR.Visu_Adv_Arr[6] := FALSE;
   TL_EXTN_UNIT_ERR.Visu_Adv_Arr[7] := FALSE;
   TL_EXTN_UNIT_ERR.Visu_Adv_Arr[8] := FALSE;
   TL_EXTN_UNIT_ERR.Visu_Adv_Arr[9] := FALSE;
   TL_EXTN_UNIT_ERR.Visu_Adv_Arr[10] := FALSE;
   TL_EXTN_UNIT_ERR.Visu_Adv_Arr[11] := FALSE;
   TL_EXTN_UNIT_ERR.Visu_Adv_Arr[12] := FALSE;
   TL_EXTN_UNIT_ERR.Visu_Adv_Arr[13] := FALSE;
   TL_EXTN_UNIT_ERR.Visu_Adv_Arr[14] := FALSE;
   TL_EXTN_UNIT_ERR.Visu_Adv_Arr[15] := FALSE;
   TL_EXTN_UNIT_ERR.Visu_Ret_Arr[0] := FALSE;
   TL_EXTN_UNIT_ERR.Visu_Ret_Arr[1] := FALSE;
   TL_EXTN_UNIT_ERR.Visu_Ret_Arr[2] := FALSE;
   TL_EXTN_UNIT_ERR.Visu_Ret_Arr[3] := FALSE;
   TL_EXTN_UNIT_ERR.Visu_Ret_Arr[4] := FALSE;
   TL_EXTN_UNIT_ERR.Visu_Ret_Arr[5] := FALSE;
   TL_EXTN_UNIT_ERR.Visu_Ret_Arr[6] := FALSE;
   TL_EXTN_UNIT_ERR.Visu_Ret_Arr[7] := FALSE;
   TL_EXTN_UNIT_ERR.Visu_Ret_Arr[8] := FALSE;
   TL_EXTN_UNIT_ERR.Visu_Ret_Arr[9] := FALSE;
   TL_EXTN_UNIT_ERR.Visu_Ret_Arr[10] := FALSE;
   TL_EXTN_UNIT_ERR.Visu_Ret_Arr[11] := FALSE;
   TL_EXTN_UNIT_ERR.Visu_Ret_Arr[12] := FALSE;
   TL_EXTN_UNIT_ERR.Visu_Ret_Arr[13] := FALSE;
   TL_EXTN_UNIT_ERR.Visu_Ret_Arr[14] := FALSE;
   TL_EXTN_UNIT_ERR.Visu_Ret_Arr[15] := FALSE;
   TL_EXTN_UNIT_ERR.BLK_Move_Ret := 0;
   TL_EXTN_UNIT_ERR.Enable := FALSE;
   TL_EXTN_UNIT_ERR.Adv_End := FALSE;
   TL_EXTN_UNIT_ERR.Ret_End := FALSE;
   TL_EXTN_ADV_RET_ERR.Enable_Aux := FALSE;
   TL_EXTN_ADV_RET_ERR.Adv_Amount := 0;
   TL_EXTN_ADV_RET_ERR.Ret_Amount := 0;
   TL_EXTN_ADV_RET_ERR.LS_Adv1 := FALSE;
   TL_EXTN_ADV_RET_ERR.LS_Ret1 := FALSE;
   TL_EXTN_ADV_RET_ERR.LS_Adv2 := FALSE;
   TL_EXTN_ADV_RET_ERR.LS_Ret2 := FALSE;
   TL_EXTN_ADV_RET_ERR.LS_Adv3 := FALSE;
   TL_EXTN_ADV_RET_ERR.LS_Ret3 := FALSE;
   TL_EXTN_ADV_RET_ERR.LS_Adv4 := FALSE;
   TL_EXTN_ADV_RET_ERR.LS_Ret4 := FALSE;
   TL_EXTN_ADV_RET_ERR.SOL_Adv := FALSE;
   TL_EXTN_ADV_RET_ERR.SOL_Ret := FALSE;
   TL_EXTN_ADV_RET_ERR.M_Ready := FALSE;
   TL_EXTN_ADV_RET_ERR.T_CHK1 := T#0MS;
   TL_EXTN_ADV_RET_ERR.T_CHK2 := T#0MS;
   TL_EXTN_ADV_RET_ERR.PB_Lamp_CHK := FALSE;
   TL_EXTN_ADV_RET_ERR.PB_Error_Rst := FALSE;
   TL_EXTN_ADV_RET_ERR.M_FLICK := FALSE;
   TL_EXTN_ADV_RET_ERR.M_Adv_Err := FALSE;
   TL_EXTN_ADV_RET_ERR.M_Ret_Err := FALSE;
   TL_EXTN_ADV_RET_ERR.LP_Adv := FALSE;
   TL_EXTN_ADV_RET_ERR.LP_Ret := FALSE;
   TL_EXTN_ADV_RET_ERR.Visu_Adv := W#16#0;
   TL_EXTN_ADV_RET_ERR.Visu_Ret := W#16#0;
   TL_EXTN_ADV_RET_ERR.Error_T1.IN := FALSE;
   TL_EXTN_ADV_RET_ERR.Error_T1.PT := T#0MS;
   TL_EXTN_ADV_RET_ERR.Error_T1.Q := FALSE;
   TL_EXTN_ADV_RET_ERR.Error_T1.ET := T#0MS;
   TL_EXTN_ADV_RET_ERR.Error_T1.STATE := B#16#0;
   TL_EXTN_ADV_RET_ERR.Error_T1.STIME := T#0MS;
   TL_EXTN_ADV_RET_ERR.Error_T1.ATIME := T#0MS;
   TL_EXTN_ADV_RET_ERR.Error_T2.IN := FALSE;
   TL_EXTN_ADV_RET_ERR.Error_T2.PT := T#0MS;
   TL_EXTN_ADV_RET_ERR.Error_T2.Q := FALSE;
   TL_EXTN_ADV_RET_ERR.Error_T2.ET := T#0MS;
   TL_EXTN_ADV_RET_ERR.Error_T2.STATE := B#16#0;
   TL_EXTN_ADV_RET_ERR.Error_T2.STIME := T#0MS;
   TL_EXTN_ADV_RET_ERR.Error_T2.ATIME := T#0MS;
   TL_EXTN_ADV_RET_ERR.CHK_Aux1 := FALSE;
   TL_EXTN_ADV_RET_ERR.CHK_Aux2 := FALSE;
   TL_EXTN_ADV_RET_ERR.Error_T1_DN := FALSE;
   TL_EXTN_ADV_RET_ERR.Error_T2_DN := FALSE;
   TL_EXTN_ADV_RET_ERR.Adv_Memo := FALSE;
   TL_EXTN_ADV_RET_ERR.Visu_Adv_Arr[0] := FALSE;
   TL_EXTN_ADV_RET_ERR.Visu_Adv_Arr[1] := FALSE;
   TL_EXTN_ADV_RET_ERR.Visu_Adv_Arr[2] := FALSE;
   TL_EXTN_ADV_RET_ERR.Visu_Adv_Arr[3] := FALSE;
   TL_EXTN_ADV_RET_ERR.Visu_Adv_Arr[4] := FALSE;
   TL_EXTN_ADV_RET_ERR.Visu_Adv_Arr[5] := FALSE;
   TL_EXTN_ADV_RET_ERR.Visu_Adv_Arr[6] := FALSE;
   TL_EXTN_ADV_RET_ERR.Visu_Adv_Arr[7] := FALSE;
   TL_EXTN_ADV_RET_ERR.Visu_Adv_Arr[8] := FALSE;
   TL_EXTN_ADV_RET_ERR.Visu_Adv_Arr[9] := FALSE;
   TL_EXTN_ADV_RET_ERR.Visu_Adv_Arr[10] := FALSE;
   TL_EXTN_ADV_RET_ERR.Visu_Adv_Arr[11] := FALSE;
   TL_EXTN_ADV_RET_ERR.Visu_Adv_Arr[12] := FALSE;
   TL_EXTN_ADV_RET_ERR.Visu_Adv_Arr[13] := FALSE;
   TL_EXTN_ADV_RET_ERR.Visu_Adv_Arr[14] := FALSE;
   TL_EXTN_ADV_RET_ERR.Visu_Adv_Arr[15] := FALSE;
   TL_EXTN_ADV_RET_ERR.Visu_Ret_Arr[0] := FALSE;
   TL_EXTN_ADV_RET_ERR.Visu_Ret_Arr[1] := FALSE;
   TL_EXTN_ADV_RET_ERR.Visu_Ret_Arr[2] := FALSE;
   TL_EXTN_ADV_RET_ERR.Visu_Ret_Arr[3] := FALSE;
   TL_EXTN_ADV_RET_ERR.Visu_Ret_Arr[4] := FALSE;
   TL_EXTN_ADV_RET_ERR.Visu_Ret_Arr[5] := FALSE;
   TL_EXTN_ADV_RET_ERR.Visu_Ret_Arr[6] := FALSE;
   TL_EXTN_ADV_RET_ERR.Visu_Ret_Arr[7] := FALSE;
   TL_EXTN_ADV_RET_ERR.Visu_Ret_Arr[8] := FALSE;
   TL_EXTN_ADV_RET_ERR.Visu_Ret_Arr[9] := FALSE;
   TL_EXTN_ADV_RET_ERR.Visu_Ret_Arr[10] := FALSE;
   TL_EXTN_ADV_RET_ERR.Visu_Ret_Arr[11] := FALSE;
   TL_EXTN_ADV_RET_ERR.Visu_Ret_Arr[12] := FALSE;
   TL_EXTN_ADV_RET_ERR.Visu_Ret_Arr[13] := FALSE;
   TL_EXTN_ADV_RET_ERR.Visu_Ret_Arr[14] := FALSE;
   TL_EXTN_ADV_RET_ERR.Visu_Ret_Arr[15] := FALSE;
   TL_EXTN_ADV_RET_ERR.BLK_Move_Ret := 0;
   TL_EXTN_ADV_RET_ERR.Enable := FALSE;
   TL_EXTN_ADV_RET_ERR.Adv_End := FALSE;
   TL_EXTN_ADV_RET_ERR.Ret_End := FALSE;
END_DATA_BLOCK

FUNCTION FC 131 : VOID
TITLE =
VERSION : 0.1

BEGIN
NETWORK
TITLE =
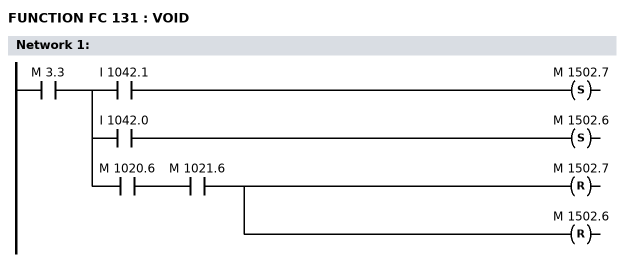

      A     M      3.3;
      =     L      0.0;
      A     L      0.0;
      A     I   1042.1;
      S     M   1502.7;
      A     L      0.0;
      A     I   1042.0;
      S     M   1502.6;
      A     L      0.0;
      A     M   1020.6;
      A     M   1021.6;
      R     M   1502.7;
      R     M   1502.6;
END_FUNCTION

FUNCTION_BLOCK FB 132
TITLE =
VERSION : 0.1

BEGIN
NETWORK
TITLE =
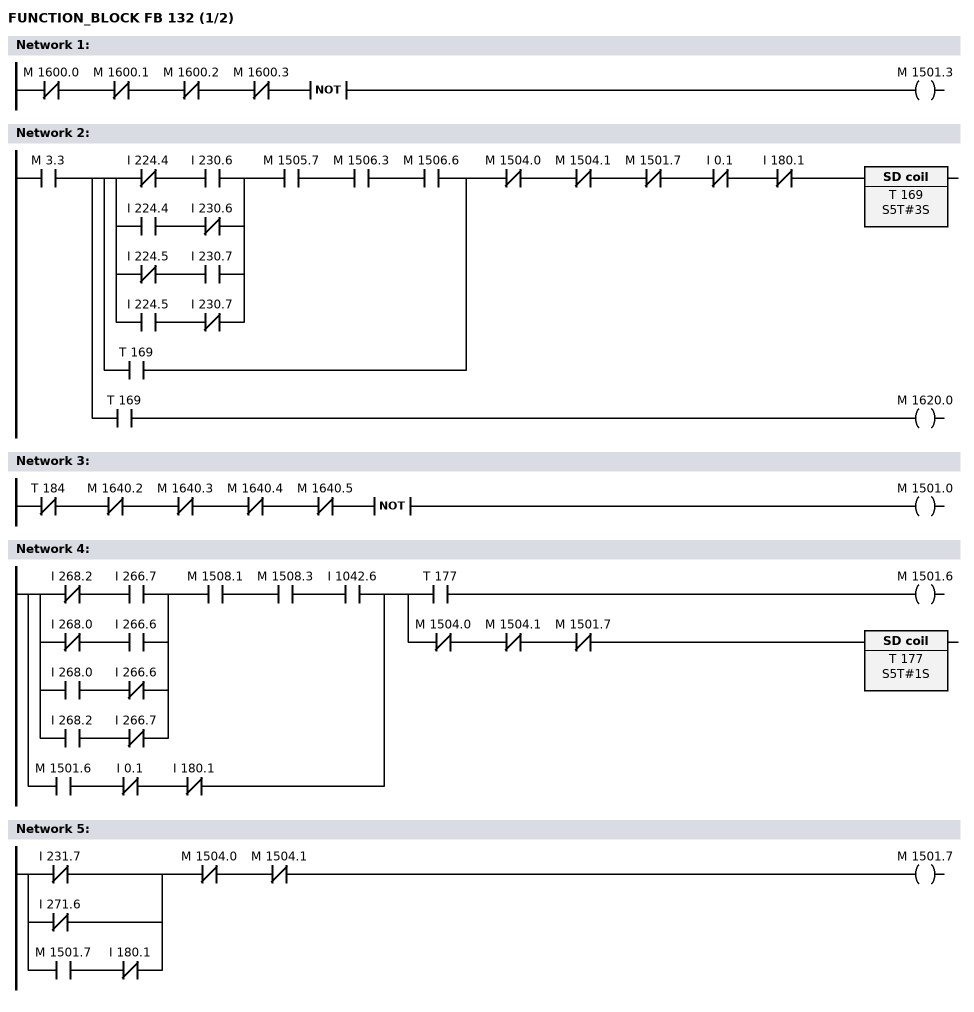

      AN    M   1600.0;
      AN    M   1600.1;
      AN    M   1600.2;
      AN    M   1600.3;
      NOT   ;
      =     M   1501.3;
NETWORK
TITLE =

      A     M      3.3;
      =     L      0.0;
      A     L      0.0;
      A(    ;
      A(    ;
      AN    I    224.4;
      A     I    230.6;
      O     ;
      A     I    224.4;
      AN    I    230.6;
      O     ;
      AN    I    224.5;
      A     I    230.7;
      O     ;
      A     I    224.5;
      AN    I    230.7;
      )     ;
      A     M   1505.7;
      A     M   1506.3;
      A     M   1506.6;
      O     T    169;
      )     ;
      AN    M   1504.0;
      AN    M   1504.1;
      AN    M   1501.7;
      AN    I      0.1;
      AN    I    180.1;
      L     S5T#3S;
      SD    T    169;
      A     L      0.0;
      A     T    169;
      =     M   1620.0;
NETWORK
TITLE =

      AN    T    184;
      AN    M   1640.2;
      AN    M   1640.3;
      AN    M   1640.4;
      AN    M   1640.5;
      NOT   ;
      =     M   1501.0;
NETWORK
TITLE =

      A(    ;
      AN    I    268.2;
      A     I    266.7;
      O     ;
      AN    I    268.0;
      A     I    266.6;
      O     ;
      A     I    268.0;
      AN    I    266.6;
      O     ;
      A     I    268.2;
      AN    I    266.7;
      )     ;
      A     M   1508.1;
      A     M   1508.3;
      A     I   1042.6;
      O     ;
      A     M   1501.6;
      AN    I      0.1;
      AN    I    180.1;
      =     L      0.0;
      A     L      0.0;
      A     T    177;
      =     M   1501.6;
      A     L      0.0;
      AN    M   1504.0;
      AN    M   1504.1;
      AN    M   1501.7;
      L     S5T#1S;
      SD    T    177;
NETWORK
TITLE =

      A(    ;
      ON    I    231.7;
      ON    I    271.6;
      O     ;
      A     M   1501.7;
      AN    I    180.1;
      )     ;
      AN    M   1504.0;
      AN    M   1504.1;
      =     M   1501.7;
NETWORK
TITLE =
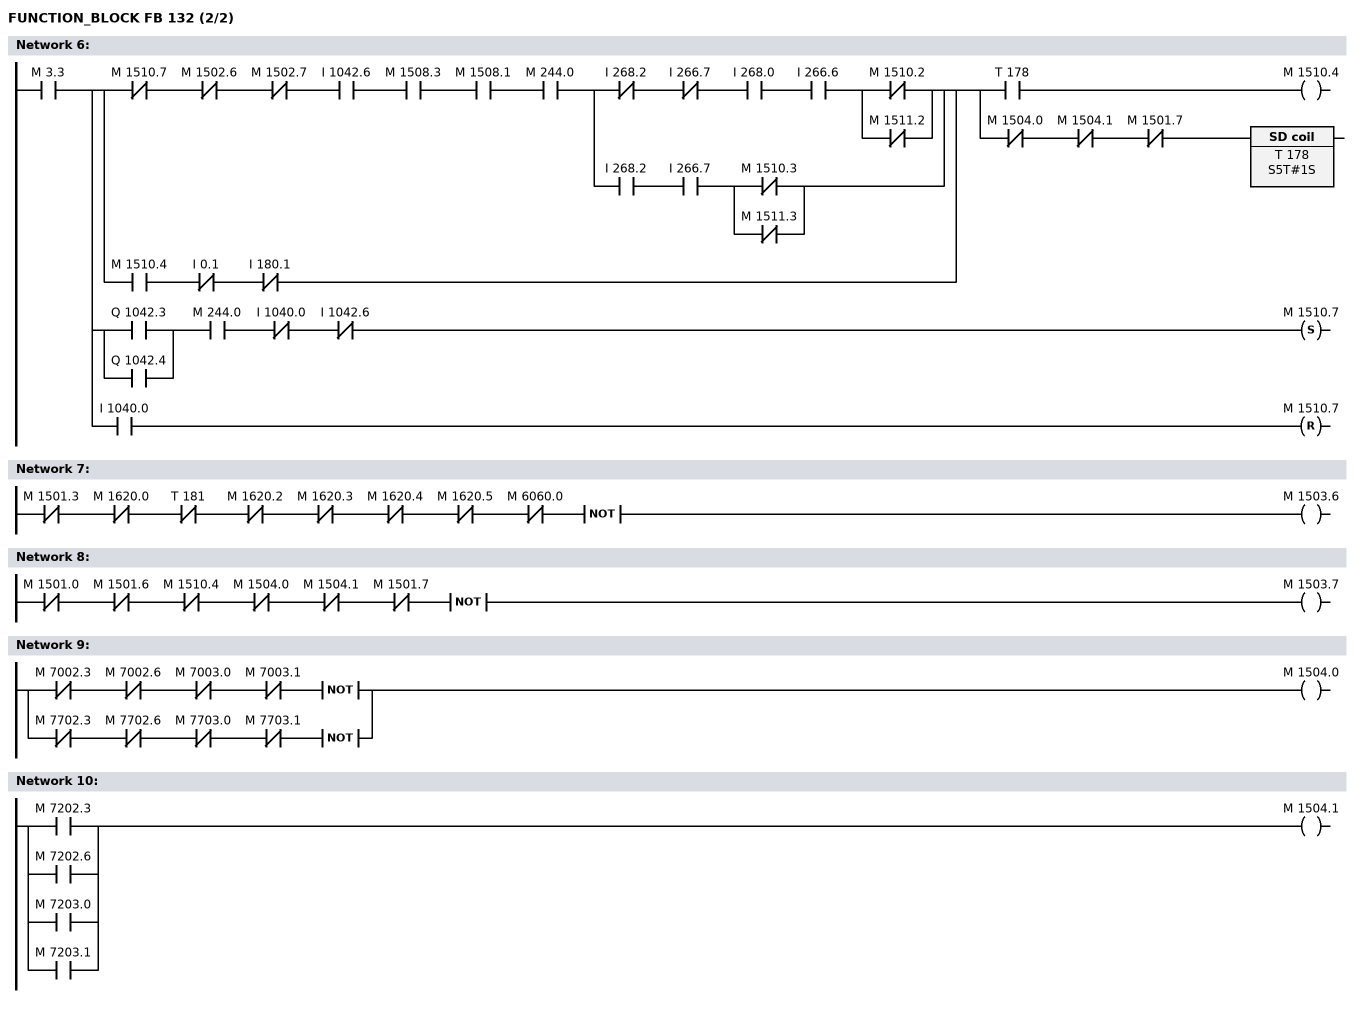

      A     M      3.3;
      =     L      0.0;
      A     L      0.0;
      A(    ;
      AN    M   1510.7;
      AN    M   1502.6;
      AN    M   1502.7;
      A     I   1042.6;
      A     M   1508.3;
      A     M   1508.1;
      A     M    244.0;
      A(    ;
      AN    I    268.2;
      AN    I    266.7;
      A     I    268.0;
      A     I    266.6;
      A(    ;
      ON    M   1510.2;
      ON    M   1511.2;
      )     ;
      O     ;
      A     I    268.2;
      A     I    266.7;
      A(    ;
      ON    M   1510.3;
      ON    M   1511.3;
      )     ;
      )     ;
      O     ;
      A     M   1510.4;
      AN    I      0.1;
      AN    I    180.1;
      )     ;
      =     L      0.1;
      A     L      0.1;
      A     T    178;
      =     M   1510.4;
      A     L      0.1;
      AN    M   1504.0;
      AN    M   1504.1;
      AN    M   1501.7;
      L     S5T#1S;
      SD    T    178;
      A     L      0.0;
      A(    ;
      O     Q   1042.3;
      O     Q   1042.4;
      )     ;
      A     M    244.0;
      AN    I   1040.0;
      AN    I   1042.6;
      S     M   1510.7;
      A     L      0.0;
      A     I   1040.0;
      R     M   1510.7;
NETWORK
TITLE =

      AN    M   1501.3;
      AN    M   1620.0;
      AN    T    181;
      AN    M   1620.2;
      AN    M   1620.3;
      AN    M   1620.4;
      AN    M   1620.5;
      AN    M   6060.0;
      NOT   ;
      =     M   1503.6;
NETWORK
TITLE =

      AN    M   1501.0;
      AN    M   1501.6;
      AN    M   1510.4;
      AN    M   1504.0;
      AN    M   1504.1;
      AN    M   1501.7;
      NOT   ;
      =     M   1503.7;
NETWORK
TITLE =

      AN    M   7002.3;
      AN    M   7002.6;
      AN    M   7003.0;
      AN    M   7003.1;
      NOT   ;
      O(    ;
      AN    M   7702.3;
      AN    M   7702.6;
      AN    M   7703.0;
      AN    M   7703.1;
      NOT   ;
      )     ;
      =     M   1504.0;
NETWORK
TITLE =

      O     M   7202.3;
      O     M   7202.6;
      O     M   7203.0;
      O     M   7203.1;
      =     M   1504.1;
END_FUNCTION_BLOCK

DATA_BLOCK DB 132
TITLE =
VERSION : 0.0

 FB 132
BEGIN
END_DATA_BLOCK

FUNCTION FC 132 : VOID
TITLE =
VERSION : 0.1

BEGIN
NETWORK
TITLE =

NETWORK
TITLE =
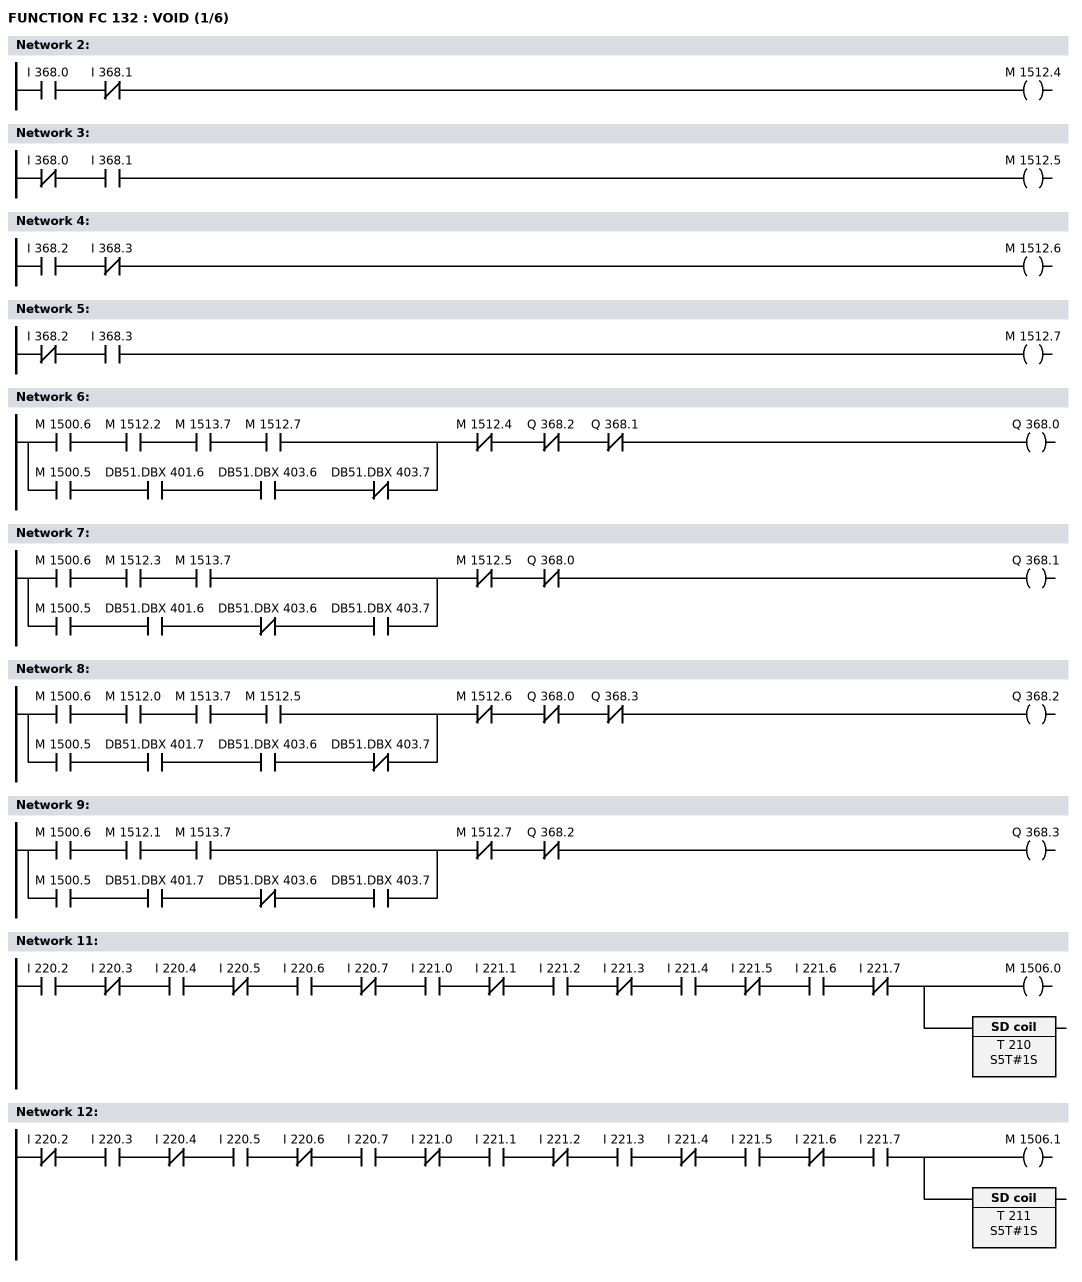

      A     I    368.0;
      AN    I    368.1;
      =     M   1512.4;
NETWORK
TITLE =

      AN    I    368.0;
      A     I    368.1;
      =     M   1512.5;
NETWORK
TITLE =

      A     I    368.2;
      AN    I    368.3;
      =     M   1512.6;
NETWORK
TITLE =

      AN    I    368.2;
      A     I    368.3;
      =     M   1512.7;
NETWORK
TITLE =

      A(    ;
      A     M   1500.6;
      A     M   1512.2;
      A     M   1513.7;
      A     M   1512.7;
      O     ;
      A     M   1500.5;
      A     DB51.DBX  401.6;
      A     DB51.DBX  403.6;
      AN    DB51.DBX  403.7;
      )     ;
      AN    M   1512.4;
      AN    Q    368.2;
      AN    Q    368.1;
      =     Q    368.0;
NETWORK
TITLE =

      A(    ;
      A     M   1500.6;
      A     M   1512.3;
      A     M   1513.7;
      O     ;
      A     M   1500.5;
      A     DB51.DBX  401.6;
      AN    DB51.DBX  403.6;
      A     DB51.DBX  403.7;
      )     ;
      AN    M   1512.5;
      AN    Q    368.0;
      =     Q    368.1;
NETWORK
TITLE =

      A(    ;
      A     M   1500.6;
      A     M   1512.0;
      A     M   1513.7;
      A     M   1512.5;
      O     ;
      A     M   1500.5;
      A     DB51.DBX  401.7;
      A     DB51.DBX  403.6;
      AN    DB51.DBX  403.7;
      )     ;
      AN    M   1512.6;
      AN    Q    368.0;
      AN    Q    368.3;
      =     Q    368.2;
NETWORK
TITLE =

      A(    ;
      A     M   1500.6;
      A     M   1512.1;
      A     M   1513.7;
      O     ;
      A     M   1500.5;
      A     DB51.DBX  401.7;
      AN    DB51.DBX  403.6;
      A     DB51.DBX  403.7;
      )     ;
      AN    M   1512.7;
      AN    Q    368.2;
      =     Q    368.3;
NETWORK
TITLE =LM EXT'N 스토리지

NETWORK
TITLE =

      A     I    220.2;
      AN    I    220.3;
      A     I    220.4;
      AN    I    220.5;
      A     I    220.6;
      AN    I    220.7;
      A     I    221.0;
      AN    I    221.1;
      A     I    221.2;
      AN    I    221.3;
      A     I    221.4;
      AN    I    221.5;
      A     I    221.6;
      AN    I    221.7;
      =     M   1506.0;
      L     S5T#1S;
      SD    T    210;
NETWORK
TITLE =

      AN    I    220.2;
      A     I    220.3;
      AN    I    220.4;
      A     I    220.5;
      AN    I    220.6;
      A     I    220.7;
      AN    I    221.0;
      A     I    221.1;
      AN    I    221.2;
      A     I    221.3;
      AN    I    221.4;
      A     I    221.5;
      AN    I    221.6;
      A     I    221.7;
      =     M   1506.1;
      L     S5T#1S;
      SD    T    211;
NETWORK
TITLE =
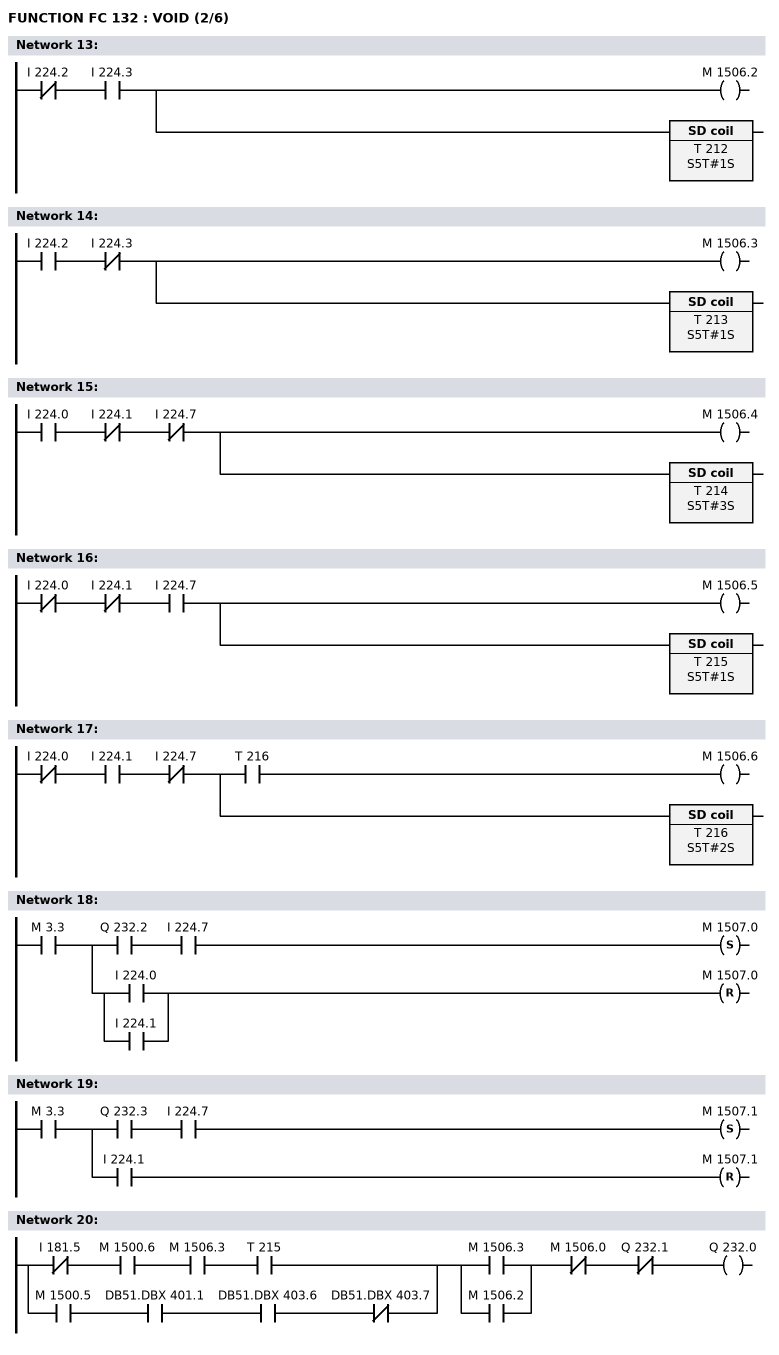

      AN    I    224.2;
      A     I    224.3;
      =     M   1506.2;
      L     S5T#1S;
      SD    T    212;
NETWORK
TITLE =

      A     I    224.2;
      AN    I    224.3;
      =     M   1506.3;
      L     S5T#1S;
      SD    T    213;
NETWORK
TITLE =

      A     I    224.0;
      AN    I    224.1;
      AN    I    224.7;
      =     M   1506.4;
      L     S5T#3S;
      SD    T    214;
NETWORK
TITLE =

      AN    I    224.0;
      AN    I    224.1;
      A     I    224.7;
      =     M   1506.5;
      L     S5T#1S;
      SD    T    215;
NETWORK
TITLE =

      AN    I    224.0;
      A     I    224.1;
      AN    I    224.7;
      =     L      0.0;
      A     L      0.0;
      A     T    216;
      =     M   1506.6;
      A     L      0.0;
      BLD   102;
      L     S5T#2S;
      SD    T    216;
NETWORK
TITLE =

      A     M      3.3;
      =     L      0.0;
      A     L      0.0;
      A     Q    232.2;
      A     I    224.7;
      S     M   1507.0;
      A     L      0.0;
      A(    ;
      O     I    224.0;
      O     I    224.1;
      )     ;
      R     M   1507.0;
NETWORK
TITLE =

      A     M      3.3;
      =     L      0.0;
      A     L      0.0;
      A     Q    232.3;
      A     I    224.7;
      S     M   1507.1;
      A     L      0.0;
      A     I    224.1;
      R     M   1507.1;
NETWORK
TITLE =

      A(    ;
      AN    I    181.5;
      A     M   1500.6;
      A     M   1506.3;
      A     T    215;
      O     ;
      A     M   1500.5;
      A     DB51.DBX  401.1;
      A     DB51.DBX  403.6;
      AN    DB51.DBX  403.7;
      )     ;
      A(    ;
      O     M   1506.3;
      O     M   1506.2;
      )     ;
      AN    M   1506.0;
      AN    Q    232.1;
      =     Q    232.0;
NETWORK
TITLE =
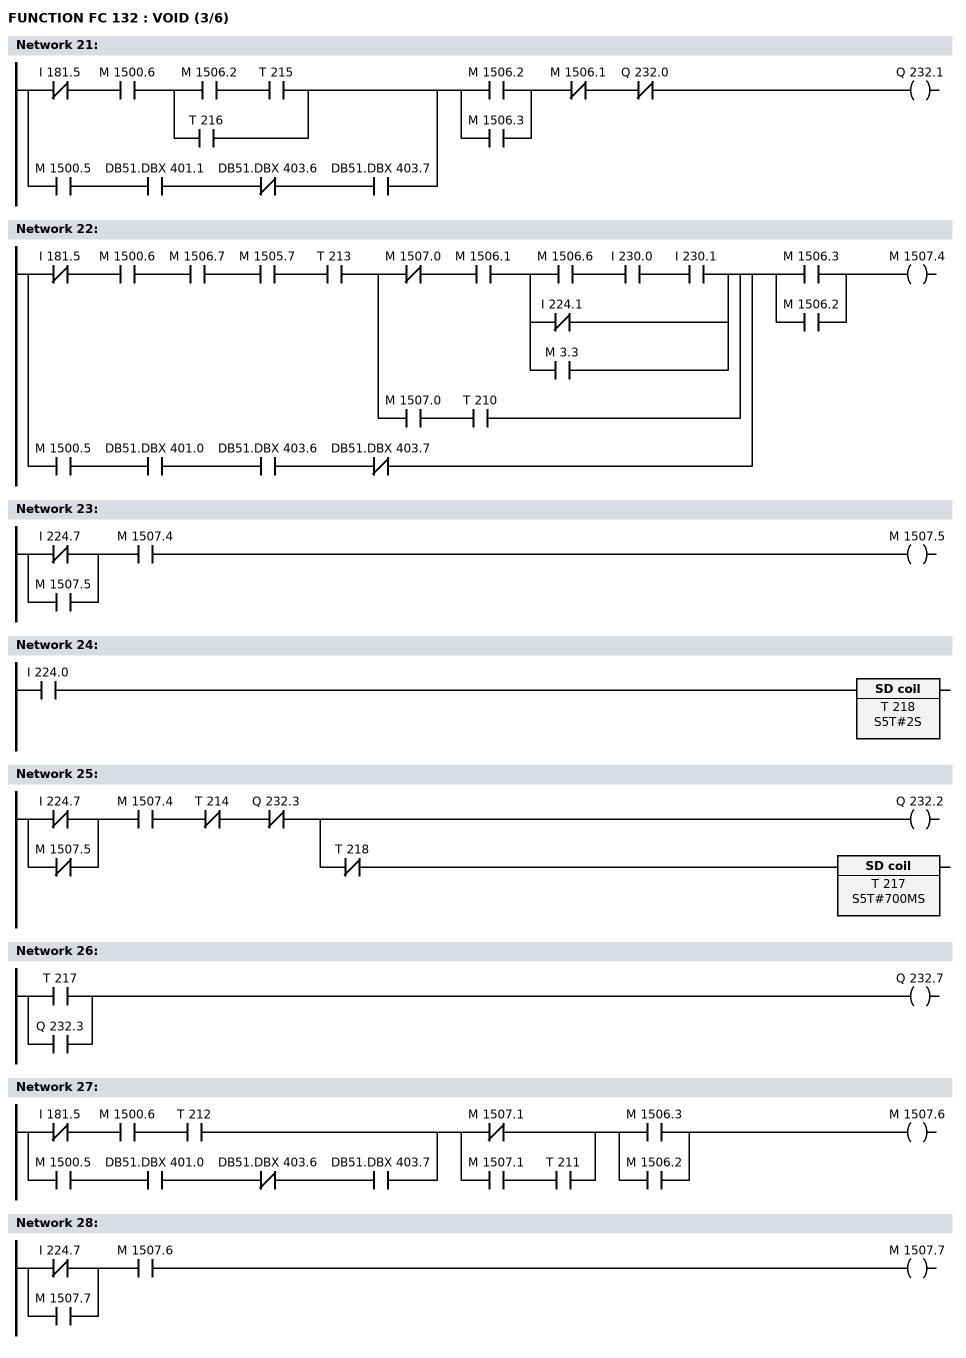

      A(    ;
      AN    I    181.5;
      A     M   1500.6;
      A(    ;
      A     M   1506.2;
      A     T    215;
      O     T    216;
      )     ;
      O     ;
      A     M   1500.5;
      A     DB51.DBX  401.1;
      AN    DB51.DBX  403.6;
      A     DB51.DBX  403.7;
      )     ;
      A(    ;
      O     M   1506.2;
      O     M   1506.3;
      )     ;
      AN    M   1506.1;
      AN    Q    232.0;
      =     Q    232.1;
NETWORK
TITLE =

      A(    ;
      AN    I    181.5;
      A     M   1500.6;
      A     M   1506.7;
      A     M   1505.7;
      A     T    213;
      A(    ;
      AN    M   1507.0;
      A     M   1506.1;
      A(    ;
      A     M   1506.6;
      A     I    230.0;
      A     I    230.1;
      ON    I    224.1;
      O     M      3.3;
      )     ;
      O     ;
      A     M   1507.0;
      A     T    210;
      )     ;
      O     ;
      A     M   1500.5;
      A     DB51.DBX  401.0;
      A     DB51.DBX  403.6;
      AN    DB51.DBX  403.7;
      )     ;
      A(    ;
      O     M   1506.3;
      O     M   1506.2;
      )     ;
      =     M   1507.4;
NETWORK
TITLE =

      A(    ;
      ON    I    224.7;
      O     M   1507.5;
      )     ;
      A     M   1507.4;
      =     M   1507.5;
NETWORK
TITLE =

      A     I    224.0;
      L     S5T#2S;
      SD    T    218;
NETWORK
TITLE =

      A(    ;
      ON    I    224.7;
      ON    M   1507.5;
      )     ;
      A     M   1507.4;
      AN    T    214;
      AN    Q    232.3;
      =     L      0.0;
      A     L      0.0;
      BLD   102;
      =     Q    232.2;
      A     L      0.0;
      AN    T    218;
      L     S5T#700MS;
      SD    T    217;
NETWORK
TITLE =

      O     T    217;
      O     Q    232.3;
      =     Q    232.7;
NETWORK
TITLE =

      A(    ;
      AN    I    181.5;
      A     M   1500.6;
      A     T    212;
      O     ;
      A     M   1500.5;
      A     DB51.DBX  401.0;
      AN    DB51.DBX  403.6;
      A     DB51.DBX  403.7;
      )     ;
      A(    ;
      ON    M   1507.1;
      O     ;
      A     M   1507.1;
      A     T    211;
      )     ;
      A(    ;
      O     M   1506.3;
      O     M   1506.2;
      )     ;
      =     M   1507.6;
NETWORK
TITLE =

      A(    ;
      ON    I    224.7;
      O     M   1507.7;
      )     ;
      A     M   1507.6;
      =     M   1507.7;
NETWORK
TITLE =
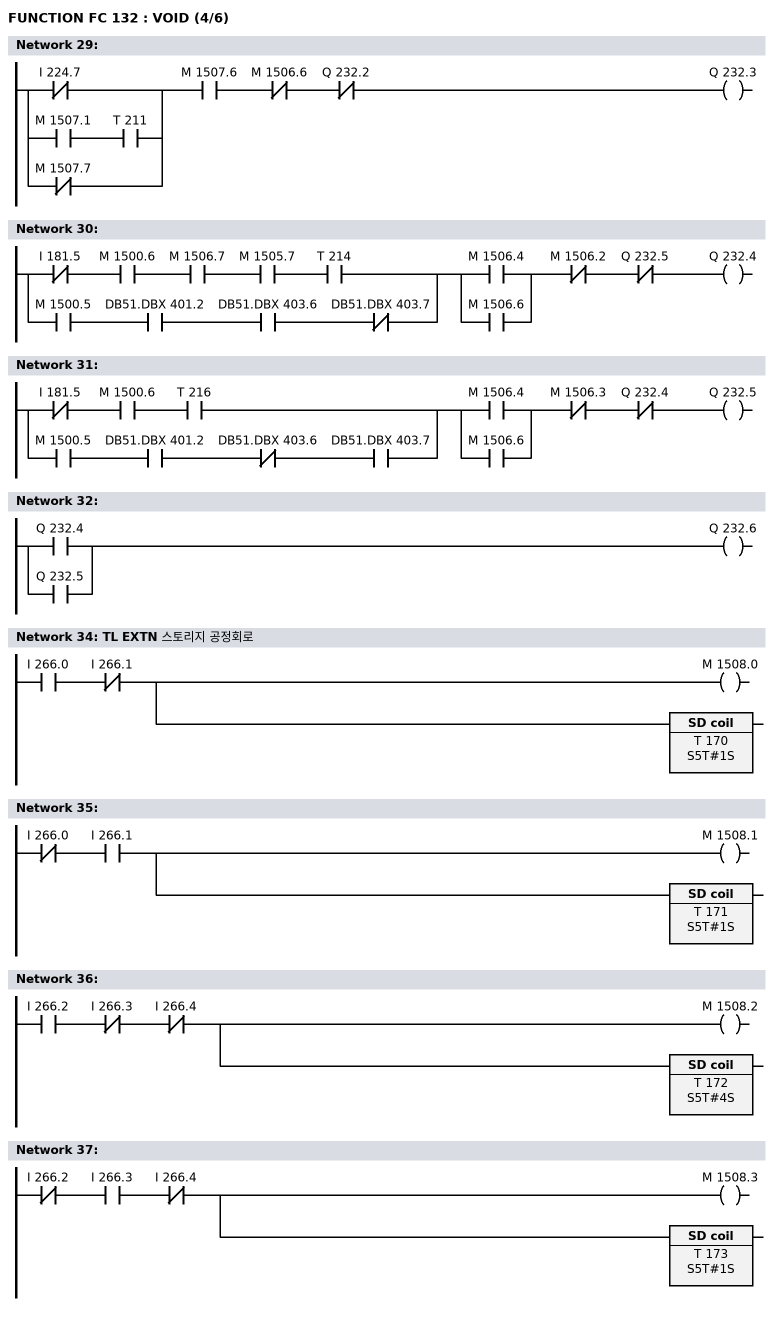

      A(    ;
      ON    I    224.7;
      O     ;
      A     M   1507.1;
      A     T    211;
      ON    M   1507.7;
      )     ;
      A     M   1507.6;
      AN    M   1506.6;
      AN    Q    232.2;
      =     Q    232.3;
NETWORK
TITLE =

      A(    ;
      AN    I    181.5;
      A     M   1500.6;
      A     M   1506.7;
      A     M   1505.7;
      A     T    214;
      O     ;
      A     M   1500.5;
      A     DB51.DBX  401.2;
      A     DB51.DBX  403.6;
      AN    DB51.DBX  403.7;
      )     ;
      A(    ;
      O     M   1506.4;
      O     M   1506.6;
      )     ;
      AN    M   1506.2;
      AN    Q    232.5;
      =     Q    232.4;
NETWORK
TITLE =

      A(    ;
      AN    I    181.5;
      A     M   1500.6;
      A     T    216;
      O     ;
      A     M   1500.5;
      A     DB51.DBX  401.2;
      AN    DB51.DBX  403.6;
      A     DB51.DBX  403.7;
      )     ;
      A(    ;
      O     M   1506.4;
      O     M   1506.6;
      )     ;
      AN    M   1506.3;
      AN    Q    232.4;
      =     Q    232.5;
NETWORK
TITLE =

      O     Q    232.4;
      O     Q    232.5;
      =     Q    232.6;
NETWORK
TITLE =TL EXT'N 스토리지

NETWORK
TITLE =TL EXTN 스토리지 공정회로

      A     I    266.0;
      AN    I    266.1;
      =     M   1508.0;
      L     S5T#1S;
      SD    T    170;
NETWORK
TITLE =

      AN    I    266.0;
      A     I    266.1;
      =     M   1508.1;
      L     S5T#1S;
      SD    T    171;
NETWORK
TITLE =

      A     I    266.2;
      AN    I    266.3;
      AN    I    266.4;
      =     M   1508.2;
      L     S5T#4S;
      SD    T    172;
NETWORK
TITLE =

      AN    I    266.2;
      A     I    266.3;
      AN    I    266.4;
      =     M   1508.3;
      L     S5T#1S;
      SD    T    173;
NETWORK
TITLE =
